Staubli VAL3: XHS3023L1.dtx

public frame fPartReal = {x=0.000, y=0.000, z=0.000, rx=0.000, ry=0.000, rz=0.000, fatherId=world[0]}
public jointRx jtPark = {j1=-10.678, j2=62.119, j3=50.568, j4=-4.773, j5=72.927, j6=-11.595}
public jointRx ptRoutingPath[2001]
  [0] = {j1=-10.678, j2=62.119, j3=50.568, j4=-4.773, j5=72.927, j6=-11.595}
  [1] = {j1=-10.681, j2=62.026, j3=50.659, j4=-4.767, j5=72.852, j6=-11.673}
  [2] = {j1=-10.699, j2=61.483, j3=51.195, j4=-4.725, j5=72.405, j6=-12.130}
  [3] = {j1=-10.720, j2=60.931, j3=51.747, j4=-4.676, j5=71.941, j6=-12.602}
  [4] = {j1=-10.743, j2=60.372, j3=52.310, j4=-4.622, j5=71.468, j6=-13.083}
  [5] = {j1=-10.767, j2=59.811, j3=52.876, j4=-4.565, j5=70.997, j6=-13.564}
  [6] = {j1=-10.793, j2=59.252, j3=53.439, j4=-4.508, j5=70.539, j6=-14.037}
  [7] = {j1=-10.819, j2=58.700, j3=53.990, j4=-4.453, j5=70.102, j6=-14.493}
  [8] = {j1=-10.845, j2=58.158, j3=54.522, j4=-4.401, j5=69.700, j6=-14.925}
  [9] = {j1=-10.866, j2=57.696, j3=54.966, j4=-4.361, j5=69.383, j6=-15.276}
  [10] = {j1=-10.885, j2=57.246, j3=55.388, j4=-4.328, j5=69.100, j6=-15.601}
  [11] = {j1=-10.904, j2=56.809, j3=55.786, j4=-4.299, j5=68.851, j6=-15.902}
  [12] = {j1=-10.922, j2=56.386, j3=56.159, j4=-4.271, j5=68.636, j6=-16.181}
  [13] = {j1=-10.923, j2=56.371, j3=56.172, j4=-4.270, j5=68.629, j6=-16.191}
  [14] = {j1=-10.924, j2=56.416, j3=56.089, j4=-4.262, j5=68.750, j6=-16.121}
  [15] = {j1=-10.923, j2=56.431, j3=56.076, j4=-4.263, j5=68.757, j6=-16.111}
  [16] = {j1=-10.905, j2=56.852, j3=55.709, j4=-4.290, j5=68.965, j6=-15.836}
  [17] = {j1=-10.887, j2=57.285, j3=55.318, j4=-4.319, j5=69.205, j6=-15.540}
  [18] = {j1=-10.868, j2=57.731, j3=54.903, j4=-4.352, j5=69.480, j6=-15.220}
  [19] = {j1=-10.847, j2=58.190, j3=54.465, j4=-4.392, j5=69.790, j6=-14.873}
  [20] = {j1=-10.821, j2=58.729, j3=53.938, j4=-4.443, j5=70.187, j6=-14.445}
  [21] = {j1=-10.795, j2=59.281, j3=53.389, j4=-4.499, j5=70.621, j6=-13.990}
  [22] = {j1=-10.770, j2=59.839, j3=52.827, j4=-4.556, j5=71.079, j6=-13.517}
  [23] = {j1=-10.745, j2=60.400, j3=52.260, j4=-4.612, j5=71.551, j6=-13.035}
  [24] = {j1=-10.722, j2=60.960, j3=51.696, j4=-4.667, j5=72.026, j6=-12.553}
  [25] = {j1=-10.701, j2=61.513, j3=51.143, j4=-4.716, j5=72.492, j6=-12.079}
  [26] = {j1=-10.683, j2=62.055, j3=50.607, j4=-4.758, j5=72.939, j6=-11.621}
  [27] = {j1=-10.681, j2=62.148, j3=50.516, j4=-4.764, j5=73.014, j6=-11.544}
  [28] = {j1=-10.683, j2=62.177, j3=50.465, j4=-4.755, j5=73.100, j6=-11.493}
  [29] = {j1=-10.686, j2=62.084, j3=50.556, j4=-4.748, j5=73.025, j6=-11.570}
  [30] = {j1=-10.704, j2=61.541, j3=51.091, j4=-4.706, j5=72.577, j6=-12.029}
  [31] = {j1=-10.724, j2=60.988, j3=51.645, j4=-4.657, j5=72.110, j6=-12.504}
  [32] = {j1=-10.748, j2=60.428, j3=52.209, j4=-4.603, j5=71.634, j6=-12.987}
  [33] = {j1=-10.772, j2=59.867, j3=52.776, j4=-4.546, j5=71.162, j6=-13.470}
  [34] = {j1=-10.798, j2=59.309, j3=53.338, j4=-4.489, j5=70.704, j6=-13.942}
  [35] = {j1=-10.824, j2=58.759, j3=53.884, j4=-4.434, j5=70.274, j6=-14.396}
  [36] = {j1=-10.849, j2=58.222, j3=54.407, j4=-4.383, j5=69.882, j6=-14.821}
  [37] = {j1=-10.870, j2=57.767, j3=54.839, j4=-4.344, j5=69.580, j6=-15.164}
  [38] = {j1=-10.889, j2=57.325, j3=55.246, j4=-4.311, j5=69.314, j6=-15.478}
  [39] = {j1=-10.907, j2=56.895, j3=55.630, j4=-4.282, j5=69.082, j6=-15.769}
  [40] = {j1=-10.924, j2=56.478, j3=55.991, j4=-4.256, j5=68.881, j6=-16.040}
  [41] = {j1=-10.925, j2=56.463, j3=56.004, j4=-4.255, j5=68.874, j6=-16.050}
  [42] = {j1=-10.926, j2=56.510, j3=55.918, j4=-4.247, j5=68.999, j6=-15.977}
  [43] = {j1=-10.926, j2=56.525, j3=55.906, j4=-4.248, j5=69.006, j6=-15.968}
  [44] = {j1=-10.908, j2=56.939, j3=55.550, j4=-4.274, j5=69.200, j6=-15.701}
  [45] = {j1=-10.891, j2=57.365, j3=55.173, j4=-4.303, j5=69.423, j6=-15.415}
  [46] = {j1=-10.872, j2=57.803, j3=54.773, j4=-4.335, j5=69.680, j6=-15.106}
  [47] = {j1=-10.851, j2=58.255, j3=54.348, j4=-4.374, j5=69.975, j6=-14.768}
  [48] = {j1=-10.826, j2=58.789, j3=53.830, j4=-4.425, j5=70.361, j6=-14.346}
  [49] = {j1=-10.800, j2=59.338, j3=53.286, j4=-4.480, j5=70.788, j6=-13.894}
  [50] = {j1=-10.775, j2=59.896, j3=52.726, j4=-4.537, j5=71.245, j6=-13.422}
  [51] = {j1=-10.750, j2=60.457, j3=52.158, j4=-4.594, j5=71.719, j6=-12.939}
  [52] = {j1=-10.727, j2=61.017, j3=51.593, j4=-4.648, j5=72.196, j6=-12.455}
  [53] = {j1=-10.706, j2=61.571, j3=51.038, j4=-4.697, j5=72.665, j6=-11.979}
  [54] = {j1=-10.688, j2=62.114, j3=50.503, j4=-4.740, j5=73.113, j6=-11.519}
  [55] = {j1=-10.685, j2=62.207, j3=50.412, j4=-4.746, j5=73.189, j6=-11.442}
  [56] = {j1=-10.688, j2=62.236, j3=50.361, j4=-4.737, j5=73.274, j6=-11.391}
  [57] = {j1=-10.690, j2=62.143, j3=50.451, j4=-4.731, j5=73.199, j6=-11.468}
  [58] = {j1=-10.708, j2=61.600, j3=50.987, j4=-4.688, j5=72.750, j6=-11.929}
  [59] = {j1=-10.729, j2=61.046, j3=51.542, j4=-4.639, j5=72.280, j6=-12.406}
  [60] = {j1=-10.752, j2=60.485, j3=52.108, j4=-4.584, j5=71.802, j6=-12.892}
  [61] = {j1=-10.777, j2=59.924, j3=52.675, j4=-4.527, j5=71.329, j6=-13.375}
  [62] = {j1=-10.803, j2=59.367, j3=53.234, j4=-4.471, j5=70.873, j6=-13.847}
  [63] = {j1=-10.828, j2=58.820, j3=53.775, j4=-4.416, j5=70.449, j6=-14.296}
  [64] = {j1=-10.853, j2=58.288, j3=54.287, j4=-4.365, j5=70.069, j6=-14.715}
  [65] = {j1=-10.873, j2=57.840, j3=54.706, j4=-4.327, j5=69.783, j6=-15.048}
  [66] = {j1=-10.892, j2=57.407, j3=55.098, j4=-4.295, j5=69.536, j6=-15.351}
  [67] = {j1=-10.910, j2=56.985, j3=55.467, j4=-4.267, j5=69.322, j6=-15.632}
  [68] = {j1=-10.927, j2=56.575, j3=55.817, j4=-4.241, j5=69.134, j6=-15.895}
  [69] = {j1=-10.927, j2=56.560, j3=55.829, j4=-4.240, j5=69.128, j6=-15.904}
  [70] = {j1=-10.928, j2=56.621, j3=55.718, j4=-4.231, j5=69.288, j6=-15.811}
  [71] = {j1=-10.928, j2=56.636, j3=55.706, j4=-4.232, j5=69.295, j6=-15.802}
  [72] = {j1=-10.911, j2=57.043, j3=55.363, j4=-4.257, j5=69.474, j6=-15.544}
  [73] = {j1=-10.894, j2=57.459, j3=55.003, j4=-4.285, j5=69.677, j6=-15.270}
  [74] = {j1=-10.876, j2=57.887, j3=54.621, j4=-4.317, j5=69.912, j6=-14.974}
  [75] = {j1=-10.856, j2=58.331, j3=54.211, j4=-4.355, j5=70.188, j6=-14.647}
  [76] = {j1=-10.831, j2=58.858, j3=53.705, j4=-4.405, j5=70.560, j6=-14.233}
  [77] = {j1=-10.806, j2=59.403, j3=53.168, j4=-4.459, j5=70.980, j6=-13.786}
  [78] = {j1=-10.780, j2=59.960, j3=52.611, j4=-4.516, j5=71.434, j6=-13.315}
  [79] = {j1=-10.756, j2=60.521, j3=52.043, j4=-4.573, j5=71.908, j6=-12.832}
  [80] = {j1=-10.732, j2=61.082, j3=51.477, j4=-4.627, j5=72.388, j6=-12.345}
  [81] = {j1=-10.711, j2=61.637, j3=50.921, j4=-4.677, j5=72.859, j6=-11.866}
  [82] = {j1=-10.693, j2=62.180, j3=50.385, j4=-4.720, j5=73.309, j6=-11.405}
  [83] = {j1=-10.690, j2=62.273, j3=50.294, j4=-4.726, j5=73.385, j6=-11.327}
  [84] = {j1=-10.678, j2=62.789, j3=49.803, j4=-4.751, j5=73.783, j6=-10.910}
  [85] = {j1=-10.672, j2=63.347, j3=49.311, j4=-4.756, j5=74.142, j6=-10.500}
  [86] = {j1=-10.674, j2=63.830, j3=48.958, j4=-4.737, j5=74.322, j6=-10.212}
  [87] = {j1=-10.676, j2=64.155, j3=48.796, j4=-4.723, j5=74.301, j6=-10.076}
  [88] = {j1=-10.675, j2=64.423, j3=48.741, j4=-4.732, j5=74.135, j6=-10.011}
  [89] = {j1=-10.669, j2=64.639, j3=48.777, j4=-4.763, j5=73.844, j6=-10.010}
  [90] = {j1=-10.658, j2=64.813, j3=48.889, j4=-4.819, j5=73.445, j6=-10.061}
  [91] = {j1=-10.643, j2=64.951, j3=49.062, j4=-4.902, j5=72.957, j6=-10.154}
  [92] = {j1=-10.621, j2=65.058, j3=49.282, j4=-5.014, j5=72.397, j6=-10.276}
  [93] = {j1=-10.593, j2=65.143, j3=49.536, j4=-5.161, j5=71.781, j6=-10.416}
  [94] = {j1=-10.592, j2=65.169, j3=49.489, j4=-5.169, j5=71.871, j6=-10.348}
  [95] = {j1=-10.620, j2=65.085, j3=49.236, j4=-5.021, j5=72.484, j6=-10.211}
  [96] = {j1=-10.642, j2=64.977, j3=49.016, j4=-4.907, j5=73.043, j6=-10.091}
  [97] = {j1=-10.658, j2=64.839, j3=48.843, j4=-4.824, j5=73.530, j6=-10.001}
  [98] = {j1=-10.669, j2=64.666, j3=48.732, j4=-4.766, j5=73.927, j6=-9.952}
  [99] = {j1=-10.675, j2=64.449, j3=48.695, j4=-4.733, j5=74.218, j6=-9.955}
  [100] = {j1=-10.677, j2=64.182, j3=48.749, j4=-4.722, j5=74.384, j6=-10.021}
  [101] = {j1=-10.675, j2=63.857, j3=48.909, j4=-4.734, j5=74.406, j6=-10.160}
  [102] = {j1=-10.673, j2=63.375, j3=49.261, j4=-4.750, j5=74.227, j6=-10.449}
  [103] = {j1=-10.680, j2=62.818, j3=49.751, j4=-4.743, j5=73.869, j6=-10.860}
  [104] = {j1=-10.693, j2=62.303, j3=50.242, j4=-4.718, j5=73.472, j6=-11.278}
  [105] = {j1=-10.695, j2=62.210, j3=50.332, j4=-4.711, j5=73.397, j6=-11.355}
  [106] = {j1=-10.714, j2=61.667, j3=50.868, j4=-4.668, j5=72.946, j6=-11.818}
  [107] = {j1=-10.735, j2=61.112, j3=51.424, j4=-4.618, j5=72.474, j6=-12.297}
  [108] = {j1=-10.758, j2=60.551, j3=51.990, j4=-4.564, j5=71.994, j6=-12.785}
  [109] = {j1=-10.782, j2=59.990, j3=52.557, j4=-4.507, j5=71.521, j6=-13.268}
  [110] = {j1=-10.808, j2=59.434, j3=53.112, j4=-4.451, j5=71.068, j6=-13.738}
  [111] = {j1=-10.833, j2=58.891, j3=53.646, j4=-4.397, j5=70.652, j6=-14.183}
  [112] = {j1=-10.857, j2=58.367, j3=54.146, j4=-4.347, j5=70.288, j6=-14.593}
  [113] = {j1=-10.877, j2=57.927, j3=54.549, j4=-4.310, j5=70.020, j6=-14.915}
  [114] = {j1=-10.895, j2=57.503, j3=54.924, j4=-4.278, j5=69.794, j6=-15.206}
  [115] = {j1=-10.912, j2=57.091, j3=55.276, j4=-4.251, j5=69.600, j6=-15.475}
  [116] = {j1=-10.929, j2=56.687, j3=55.613, j4=-4.226, j5=69.428, j6=-15.729}
  [117] = {j1=-10.929, j2=56.672, j3=55.625, j4=-4.225, j5=69.422, j6=-15.738}
  [118] = {j1=-10.930, j2=56.719, j3=55.540, j4=-4.218, j5=69.545, j6=-15.666}
  [119] = {j1=-10.930, j2=56.734, j3=55.528, j4=-4.219, j5=69.551, j6=-15.657}
  [120] = {j1=-10.913, j2=57.135, j3=55.196, j4=-4.244, j5=69.717, j6=-15.407}
  [121] = {j1=-10.896, j2=57.544, j3=54.850, j4=-4.271, j5=69.904, j6=-15.143}
  [122] = {j1=-10.879, j2=57.964, j3=54.482, j4=-4.302, j5=70.122, j6=-14.856}
  [123] = {j1=-10.859, j2=58.401, j3=54.085, j4=-4.339, j5=70.383, j6=-14.539}
  [124] = {j1=-10.835, j2=58.923, j3=53.589, j4=-4.389, j5=70.742, j6=-14.133}
  [125] = {j1=-10.810, j2=59.465, j3=53.058, j4=-4.442, j5=71.155, j6=-13.690}
  [126] = {j1=-10.785, j2=60.019, j3=52.504, j4=-4.498, j5=71.606, j6=-13.221}
  [127] = {j1=-10.760, j2=60.580, j3=51.938, j4=-4.555, j5=72.079, j6=-12.737}
  [128] = {j1=-10.737, j2=61.141, j3=51.371, j4=-4.609, j5=72.560, j6=-12.250}
  [129] = {j1=-10.716, j2=61.696, j3=50.815, j4=-4.659, j5=73.034, j6=-11.769}
  [130] = {j1=-10.698, j2=62.240, j3=50.279, j4=-4.703, j5=73.485, j6=-11.306}
  [131] = {j1=-10.695, j2=62.333, j3=50.188, j4=-4.709, j5=73.560, j6=-11.228}
  [132] = {j1=-10.682, j2=62.848, j3=49.698, j4=-4.736, j5=73.958, j6=-10.810}
  [133] = {j1=-10.675, j2=63.405, j3=49.209, j4=-4.745, j5=74.315, j6=-10.398}
  [134] = {j1=-10.676, j2=63.886, j3=48.858, j4=-4.731, j5=74.494, j6=-10.107}
  [135] = {j1=-10.677, j2=64.211, j3=48.698, j4=-4.721, j5=74.472, j6=-9.966}
  [136] = {j1=-10.675, j2=64.478, j3=48.644, j4=-4.734, j5=74.307, j6=-9.898}
  [137] = {j1=-10.668, j2=64.695, j3=48.681, j4=-4.769, j5=74.017, j6=-9.893}
  [138] = {j1=-10.657, j2=64.868, j3=48.792, j4=-4.829, j5=73.621, j6=-9.940}
  [139] = {j1=-10.641, j2=65.006, j3=48.965, j4=-4.914, j5=73.136, j6=-10.029}
  [140] = {j1=-10.619, j2=65.114, j3=49.184, j4=-5.029, j5=72.580, j6=-10.147}
  [141] = {j1=-10.590, j2=65.199, j3=49.436, j4=-5.178, j5=71.969, j6=-10.281}
  [142] = {j1=-10.589, j2=65.226, j3=49.390, j4=-5.186, j5=72.057, j6=-10.214}
  [143] = {j1=-10.618, j2=65.140, j3=49.138, j4=-5.036, j5=72.666, j6=-10.082}
  [144] = {j1=-10.640, j2=65.032, j3=48.919, j4=-4.920, j5=73.222, j6=-9.966}
  [145] = {j1=-10.656, j2=64.895, j3=48.746, j4=-4.833, j5=73.706, j6=-9.880}
  [146] = {j1=-10.668, j2=64.721, j3=48.634, j4=-4.772, j5=74.102, j6=-9.835}
  [147] = {j1=-10.675, j2=64.505, j3=48.597, j4=-4.735, j5=74.391, j6=-9.842}
  [148] = {j1=-10.678, j2=64.238, j3=48.650, j4=-4.720, j5=74.556, j6=-9.911}
  [149] = {j1=-10.677, j2=63.914, j3=48.809, j4=-4.727, j5=74.579, j6=-10.054}
  [150] = {j1=-10.677, j2=63.433, j3=49.158, j4=-4.739, j5=74.401, j6=-10.347}
  [151] = {j1=-10.684, j2=62.877, j3=49.646, j4=-4.728, j5=74.044, j6=-10.760}
  [152] = {j1=-10.697, j2=62.362, j3=50.136, j4=-4.701, j5=73.647, j6=-11.179}
  [153] = {j1=-10.700, j2=62.269, j3=50.226, j4=-4.694, j5=73.572, j6=-11.257}
  [154] = {j1=-10.718, j2=61.726, j3=50.761, j4=-4.651, j5=73.121, j6=-11.721}
  [155] = {j1=-10.739, j2=61.171, j3=51.318, j4=-4.601, j5=72.648, j6=-12.202}
  [156] = {j1=-10.762, j2=60.611, j3=51.883, j4=-4.546, j5=72.168, j6=-12.690}
  [157] = {j1=-10.787, j2=60.050, j3=52.448, j4=-4.490, j5=71.696, j6=-13.173}
  [158] = {j1=-10.812, j2=59.497, j3=53.000, j4=-4.434, j5=71.247, j6=-13.641}
  [159] = {j1=-10.837, j2=58.957, j3=53.527, j4=-4.381, j5=70.838, j6=-14.082}
  [160] = {j1=-10.861, j2=58.438, j3=54.018, j4=-4.332, j5=70.485, j6=-14.484}
  [161] = {j1=-10.880, j2=58.005, j3=54.409, j4=-4.295, j5=70.232, j6=-14.797}
  [162] = {j1=-10.897, j2=57.588, j3=54.770, j4=-4.264, j5=70.022, j6=-15.079}
  [163] = {j1=-10.914, j2=57.183, j3=55.110, j4=-4.237, j5=69.842, j6=-15.340}
  [164] = {j1=-10.930, j2=56.784, j3=55.437, j4=-4.213, j5=69.681, j6=-15.587}
  [165] = {j1=-10.931, j2=56.770, j3=55.449, j4=-4.212, j5=69.676, j6=-15.596}
  [166] = {j1=-10.932, j2=56.814, j3=55.368, j4=-4.205, j5=69.793, j6=-15.527}
  [167] = {j1=-10.931, j2=56.829, j3=55.356, j4=-4.206, j5=69.799, j6=-15.518}
  [168] = {j1=-10.915, j2=57.225, j3=55.032, j4=-4.231, j5=69.956, j6=-15.273}
  [169] = {j1=-10.899, j2=57.628, j3=54.698, j4=-4.258, j5=70.130, j6=-15.017}
  [170] = {j1=-10.881, j2=58.042, j3=54.342, j4=-4.288, j5=70.334, j6=-14.739}
  [171] = {j1=-10.862, j2=58.473, j3=53.955, j4=-4.325, j5=70.582, j6=-14.429}
  [172] = {j1=-10.839, j2=58.990, j3=53.469, j4=-4.373, j5=70.930, j6=-14.030}
  [173] = {j1=-10.814, j2=59.528, j3=52.944, j4=-4.426, j5=71.336, j6=-13.592}
  [174] = {j1=-10.789, j2=60.081, j3=52.394, j4=-4.481, j5=71.783, j6=-13.125}
  [175] = {j1=-10.765, j2=60.641, j3=51.830, j4=-4.537, j5=72.255, j6=-12.642}
  [176] = {j1=-10.741, j2=61.201, j3=51.264, j4=-4.592, j5=72.735, j6=-12.154}
  [177] = {j1=-10.720, j2=61.756, j3=50.708, j4=-4.642, j5=73.209, j6=-11.672}
  [178] = {j1=-10.702, j2=62.299, j3=50.173, j4=-4.686, j5=73.660, j6=-11.208}
  [179] = {j1=-10.699, j2=62.392, j3=50.082, j4=-4.693, j5=73.736, j6=-11.130}
  [180] = {j1=-10.686, j2=62.907, j3=49.593, j4=-4.721, j5=74.133, j6=-10.710}
  [181] = {j1=-10.678, j2=63.464, j3=49.105, j4=-4.733, j5=74.490, j6=-10.296}
  [182] = {j1=-10.678, j2=63.944, j3=48.756, j4=-4.725, j5=74.668, j6=-10.000}
  [183] = {j1=-10.678, j2=64.268, j3=48.597, j4=-4.720, j5=74.646, j6=-9.856}
  [184] = {j1=-10.675, j2=64.535, j3=48.545, j4=-4.737, j5=74.482, j6=-9.785}
  [185] = {j1=-10.667, j2=64.751, j3=48.582, j4=-4.776, j5=74.193, j6=-9.776}
  [186] = {j1=-10.655, j2=64.924, j3=48.694, j4=-4.838, j5=73.799, j6=-9.819}
  [187] = {j1=-10.639, j2=65.062, j3=48.867, j4=-4.927, j5=73.316, j6=-9.904}
  [188] = {j1=-10.616, j2=65.170, j3=49.085, j4=-5.044, j5=72.763, j6=-10.018}
  [189] = {j1=-10.587, j2=65.256, j3=49.337, j4=-5.196, j5=72.156, j6=-10.148}
  [190] = {j1=-10.586, j2=65.282, j3=49.292, j4=-5.204, j5=72.243, j6=-10.082}
  [191] = {j1=-10.615, j2=65.196, j3=49.040, j4=-5.051, j5=72.849, j6=-9.954}
  [192] = {j1=-10.638, j2=65.088, j3=48.821, j4=-4.932, j5=73.402, j6=-9.842}
  [193] = {j1=-10.655, j2=64.951, j3=48.648, j4=-4.843, j5=73.884, j6=-9.759}
  [194] = {j1=-10.667, j2=64.778, j3=48.535, j4=-4.779, j5=74.278, j6=-9.717}
  [195] = {j1=-10.675, j2=64.562, j3=48.497, j4=-4.738, j5=74.567, j6=-9.728}
  [196] = {j1=-10.679, j2=64.296, j3=48.549, j4=-4.719, j5=74.731, j6=-9.801}
  [197] = {j1=-10.679, j2=63.972, j3=48.706, j4=-4.721, j5=74.753, j6=-9.947}
  [198] = {j1=-10.680, j2=63.492, j3=49.054, j4=-4.728, j5=74.576, j6=-10.245}
  [199] = {j1=-10.688, j2=62.936, j3=49.541, j4=-4.714, j5=74.219, j6=-10.661}
  [200] = {j1=-10.701, j2=62.422, j3=50.030, j4=-4.685, j5=73.823, j6=-11.081}
  [201] = {j1=-10.704, j2=62.329, j3=50.120, j4=-4.678, j5=73.748, j6=-11.160}
  [202] = {j1=-10.723, j2=61.787, j3=50.654, j4=-4.634, j5=73.297, j6=-11.624}
  [203] = {j1=-10.744, j2=61.232, j3=51.210, j4=-4.583, j5=72.824, j6=-12.106}
  [204] = {j1=-10.767, j2=60.672, j3=51.774, j4=-4.529, j5=72.344, j6=-12.594}
  [205] = {j1=-10.791, j2=60.113, j3=52.336, j4=-4.473, j5=71.874, j6=-13.076}
  [206] = {j1=-10.816, j2=59.562, j3=52.884, j4=-4.418, j5=71.430, j6=-13.542}
  [207] = {j1=-10.840, j2=59.025, j3=53.405, j4=-4.366, j5=71.028, j6=-13.978}
  [208] = {j1=-10.864, j2=58.511, j3=53.886, j4=-4.318, j5=70.686, j6=-14.374}
  [209] = {j1=-10.883, j2=58.083, j3=54.268, j4=-4.282, j5=70.444, j6=-14.680}
  [210] = {j1=-10.900, j2=57.672, j3=54.618, j4=-4.252, j5=70.247, j6=-14.955}
  [211] = {j1=-10.916, j2=57.272, j3=54.948, j4=-4.225, j5=70.079, j6=-15.208}
  [212] = {j1=-10.932, j2=56.878, j3=55.267, j4=-4.201, j5=69.926, j6=-15.451}
  [213] = {j1=-10.932, j2=56.864, j3=55.279, j4=-4.200, j5=69.921, j6=-15.460}
  [214] = {j1=-10.933, j2=56.906, j3=55.202, j4=-4.193, j5=70.034, j6=-15.393}
  [215] = {j1=-10.933, j2=56.921, j3=55.190, j4=-4.194, j5=70.039, j6=-15.385}
  [216] = {j1=-10.917, j2=57.314, j3=54.873, j4=-4.218, j5=70.189, j6=-15.144}
  [217] = {j1=-10.901, j2=57.711, j3=54.547, j4=-4.245, j5=70.353, j6=-14.893}
  [218] = {j1=-10.884, j2=58.120, j3=54.200, j4=-4.275, j5=70.546, j6=-14.621}
  [219] = {j1=-10.865, j2=58.546, j3=53.823, j4=-4.310, j5=70.784, j6=-14.318}
  [220] = {j1=-10.842, j2=59.059, j3=53.345, j4=-4.358, j5=71.122, j6=-13.925}
  [221] = {j1=-10.818, j2=59.594, j3=52.827, j4=-4.409, j5=71.521, j6=-13.491}
  [222] = {j1=-10.793, j2=60.144, j3=52.281, j4=-4.464, j5=71.963, j6=-13.027}
  [223] = {j1=-10.769, j2=60.702, j3=51.720, j4=-4.520, j5=72.432, j6=-12.546}
  [224] = {j1=-10.746, j2=61.262, j3=51.156, j4=-4.575, j5=72.911, j6=-12.058}
  [225] = {j1=-10.725, j2=61.816, j3=50.601, j4=-4.625, j5=73.384, j6=-11.576}
  [226] = {j1=-10.706, j2=62.359, j3=50.066, j4=-4.670, j5=73.836, j6=-11.111}
  [227] = {j1=-10.703, j2=62.452, j3=49.976, j4=-4.677, j5=73.911, j6=-11.033}
  [228] = {j1=-10.690, j2=62.966, j3=49.488, j4=-4.707, j5=74.308, j6=-10.611}
  [229] = {j1=-10.681, j2=63.523, j3=49.001, j4=-4.722, j5=74.666, j6=-10.194}
  [230] = {j1=-10.679, j2=64.003, j3=48.653, j4=-4.719, j5=74.844, j6=-9.894}
  [231] = {j1=-10.679, j2=64.326, j3=48.495, j4=-4.719, j5=74.823, j6=-9.746}
  [232] = {j1=-10.675, j2=64.592, j3=48.444, j4=-4.740, j5=74.659, j6=-9.671}
  [233] = {j1=-10.666, j2=64.808, j3=48.482, j4=-4.782, j5=74.371, j6=-9.658}
  [234] = {j1=-10.654, j2=64.981, j3=48.595, j4=-4.848, j5=73.978, j6=-9.698}
  [235] = {j1=-10.637, j2=65.118, j3=48.768, j4=-4.939, j5=73.497, j6=-9.779}
  [236] = {j1=-10.614, j2=65.227, j3=48.987, j4=-5.059, j5=72.946, j6=-9.890}
  [237] = {j1=-10.584, j2=65.312, j3=49.239, j4=-5.213, j5=72.342, j6=-10.017}
  [238] = {j1=-10.583, j2=65.337, j3=49.194, j4=-5.221, j5=72.428, j6=-9.951}
  [239] = {j1=-10.612, j2=65.252, j3=48.942, j4=-5.066, j5=73.031, j6=-9.826}
  [240] = {j1=-10.636, j2=65.144, j3=48.722, j4=-4.945, j5=73.582, j6=-9.717}
  [241] = {j1=-10.653, j2=65.008, j3=48.548, j4=-4.852, j5=74.063, j6=-9.638}
  [242] = {j1=-10.666, j2=64.835, j3=48.435, j4=-4.785, j5=74.456, j6=-9.600}
  [243] = {j1=-10.675, j2=64.620, j3=48.395, j4=-4.741, j5=74.744, j6=-9.614}
  [244] = {j1=-10.679, j2=64.354, j3=48.446, j4=-4.718, j5=74.908, j6=-9.691}
  [245] = {j1=-10.680, j2=64.031, j3=48.603, j4=-4.716, j5=74.930, j6=-9.840}
  [246] = {j1=-10.683, j2=63.551, j3=48.950, j4=-4.717, j5=74.751, j6=-10.143}
  [247] = {j1=-10.692, j2=62.995, j3=49.436, j4=-4.699, j5=74.394, j6=-10.562}
  [248] = {j1=-10.706, j2=62.481, j3=49.924, j4=-4.669, j5=73.998, j6=-10.984}
  [249] = {j1=-10.708, j2=62.389, j3=50.014, j4=-4.662, j5=73.923, j6=-11.063}
  [250] = {j1=-10.727, j2=61.847, j3=50.547, j4=-4.617, j5=73.472, j6=-11.528}
  [251] = {j1=-10.748, j2=61.293, j3=51.101, j4=-4.566, j5=73.000, j6=-12.010}
  [252] = {j1=-10.771, j2=60.734, j3=51.663, j4=-4.512, j5=72.523, j6=-12.497}
  [253] = {j1=-10.795, j2=60.177, j3=52.221, j4=-4.456, j5=72.057, j6=-12.977}
  [254] = {j1=-10.820, j2=59.628, j3=52.764, j4=-4.402, j5=71.618, j6=-13.440}
  [255] = {j1=-10.844, j2=59.095, j3=53.279, j4=-4.350, j5=71.223, j6=-13.872}
  [256] = {j1=-10.867, j2=58.585, j3=53.753, j4=-4.304, j5=70.889, j6=-14.262}
  [257] = {j1=-10.885, j2=58.161, j3=54.126, j4=-4.269, j5=70.656, j6=-14.563}
  [258] = {j1=-10.902, j2=57.755, j3=54.469, j4=-4.239, j5=70.468, j6=-14.832}
  [259] = {j1=-10.918, j2=57.359, j3=54.791, j4=-4.213, j5=70.309, j6=-15.080}
  [260] = {j1=-10.933, j2=56.968, j3=55.105, j4=-4.189, j5=70.162, j6=-15.320}
  [261] = {j1=-10.934, j2=56.954, j3=55.116, j4=-4.188, j5=70.157, j6=-15.329}
  [262] = {j1=-10.935, j2=56.995, j3=55.043, j4=-4.181, j5=70.265, j6=-15.265}
  [263] = {j1=-10.934, j2=57.009, j3=55.031, j4=-4.182, j5=70.270, j6=-15.257}
  [264] = {j1=-10.919, j2=57.399, j3=54.719, j4=-4.207, j5=70.416, j6=-15.018}
  [265] = {j1=-10.903, j2=57.794, j3=54.399, j4=-4.233, j5=70.573, j6=-14.771}
  [266] = {j1=-10.886, j2=58.199, j3=54.059, j4=-4.262, j5=70.758, j6=-14.504}
  [267] = {j1=-10.868, j2=58.621, j3=53.689, j4=-4.297, j5=70.988, j6=-14.206}
  [268] = {j1=-10.846, j2=59.130, j3=53.218, j4=-4.343, j5=71.318, j6=-13.818}
  [269] = {j1=-10.822, j2=59.661, j3=52.705, j4=-4.394, j5=71.711, j6=-13.388}
  [270] = {j1=-10.797, j2=60.209, j3=52.164, j4=-4.448, j5=72.148, j6=-12.927}
  [271] = {j1=-10.773, j2=60.765, j3=51.607, j4=-4.503, j5=72.612, j6=-12.448}
  [272] = {j1=-10.750, j2=61.323, j3=51.047, j4=-4.558, j5=73.088, j6=-11.962}
  [273] = {j1=-10.729, j2=61.877, j3=50.494, j4=-4.609, j5=73.559, j6=-11.480}
  [274] = {j1=-10.711, j2=62.419, j3=49.961, j4=-4.654, j5=74.010, j6=-11.015}
  [275] = {j1=-10.708, j2=62.512, j3=49.870, j4=-4.661, j5=74.086, j6=-10.936}
  [276] = {j1=-10.694, j2=63.026, j3=49.383, j4=-4.692, j5=74.483, j6=-10.513}
  [277] = {j1=-10.684, j2=63.582, j3=48.896, j4=-4.711, j5=74.841, j6=-10.092}
  [278] = {j1=-10.681, j2=64.062, j3=48.549, j4=-4.713, j5=75.021, j6=-9.787}
  [279] = {j1=-10.680, j2=64.385, j3=48.392, j4=-4.718, j5=75.000, j6=-9.635}
  [280] = {j1=-10.675, j2=64.651, j3=48.341, j4=-4.743, j5=74.837, j6=-9.556}
  [281] = {j1=-10.666, j2=64.866, j3=48.381, j4=-4.789, j5=74.550, j6=-9.541}
  [282] = {j1=-10.652, j2=65.038, j3=48.495, j4=-4.858, j5=74.158, j6=-9.577}
  [283] = {j1=-10.634, j2=65.175, j3=48.669, j4=-4.952, j5=73.678, j6=-9.656}
  [284] = {j1=-10.611, j2=65.283, j3=48.889, j4=-5.074, j5=73.128, j6=-9.763}
  [285] = {j1=-10.581, j2=65.368, j3=49.141, j4=-5.230, j5=72.526, j6=-9.886}
  [286] = {j1=-10.580, j2=65.393, j3=49.098, j4=-5.238, j5=72.611, j6=-9.822}
  [287] = {j1=-10.610, j2=65.308, j3=48.844, j4=-5.081, j5=73.213, j6=-9.700}
  [288] = {j1=-10.634, j2=65.201, j3=48.623, j4=-4.957, j5=73.763, j6=-9.594}
  [289] = {j1=-10.652, j2=65.065, j3=48.448, j4=-4.862, j5=74.243, j6=-9.517}
  [290] = {j1=-10.665, j2=64.893, j3=48.333, j4=-4.792, j5=74.636, j6=-9.481}
  [291] = {j1=-10.675, j2=64.678, j3=48.292, j4=-4.744, j5=74.923, j6=-9.499}
  [292] = {j1=-10.680, j2=64.414, j3=48.342, j4=-4.717, j5=75.087, j6=-9.579}
  [293] = {j1=-10.682, j2=64.090, j3=48.498, j4=-4.710, j5=75.107, j6=-9.733}
  [294] = {j1=-10.686, j2=63.610, j3=48.845, j4=-4.706, j5=74.927, j6=-10.041}
  [295] = {j1=-10.696, j2=63.055, j3=49.331, j4=-4.685, j5=74.569, j6=-10.464}
  [296] = {j1=-10.710, j2=62.541, j3=49.818, j4=-4.653, j5=74.172, j6=-10.888}
  [297] = {j1=-10.713, j2=62.448, j3=49.908, j4=-4.646, j5=74.097, j6=-10.967}
  [298] = {j1=-10.731, j2=61.907, j3=50.440, j4=-4.600, j5=73.647, j6=-11.432}
  [299] = {j1=-10.752, j2=61.355, j3=50.991, j4=-4.549, j5=73.178, j6=-11.914}
  [300] = {j1=-10.775, j2=60.798, j3=51.549, j4=-4.495, j5=72.705, j6=-12.399}
  [301] = {j1=-10.799, j2=60.243, j3=52.104, j4=-4.440, j5=72.243, j6=-12.877}
  [302] = {j1=-10.823, j2=59.697, j3=52.642, j4=-4.386, j5=71.810, j6=-13.336}
  [303] = {j1=-10.847, j2=59.167, j3=53.151, j4=-4.336, j5=71.421, j6=-13.764}
  [304] = {j1=-10.869, j2=58.660, j3=53.618, j4=-4.290, j5=71.095, j6=-14.149}
  [305] = {j1=-10.887, j2=58.240, j3=53.985, j4=-4.256, j5=70.868, j6=-14.446}
  [306] = {j1=-10.904, j2=57.837, j3=54.321, j4=-4.227, j5=70.687, j6=-14.711}
  [307] = {j1=-10.920, j2=57.444, j3=54.639, j4=-4.201, j5=70.532, j6=-14.956}
  [308] = {j1=-10.935, j2=57.054, j3=54.949, j4=-4.177, j5=70.389, j6=-15.194}
  [309] = {j1=-10.936, j2=57.040, j3=54.960, j4=-4.176, j5=70.384, j6=-15.203}
  [310] = {j1=-10.937, j2=57.079, j3=54.891, j4=-4.170, j5=70.487, j6=-15.143}
  [311] = {j1=-10.936, j2=57.093, j3=54.879, j4=-4.171, j5=70.492, j6=-15.134}
  [312] = {j1=-10.921, j2=57.482, j3=54.569, j4=-4.195, j5=70.636, j6=-14.896}
  [313] = {j1=-10.905, j2=57.875, j3=54.253, j4=-4.221, j5=70.789, j6=-14.651}
  [314] = {j1=-10.889, j2=58.277, j3=53.918, j4=-4.250, j5=70.970, j6=-14.387}
  [315] = {j1=-10.871, j2=58.697, j3=53.553, j4=-4.283, j5=71.194, j6=-14.093}
  [316] = {j1=-10.849, j2=59.202, j3=53.088, j4=-4.328, j5=71.518, j6=-13.709}
  [317] = {j1=-10.825, j2=59.731, j3=52.581, j4=-4.378, j5=71.904, j6=-13.283}
  [318] = {j1=-10.801, j2=60.275, j3=52.045, j4=-4.432, j5=72.335, j6=-12.826}
  [319] = {j1=-10.777, j2=60.829, j3=51.493, j4=-4.487, j5=72.794, j6=-12.349}
  [320] = {j1=-10.755, j2=61.385, j3=50.937, j4=-4.541, j5=73.266, j6=-11.865}
  [321] = {j1=-10.733, j2=61.937, j3=50.387, j4=-4.592, j5=73.734, j6=-11.385}
  [322] = {j1=-10.715, j2=62.478, j3=49.856, j4=-4.637, j5=74.184, j6=-10.919}
  [323] = {j1=-10.712, j2=62.571, j3=49.765, j4=-4.645, j5=74.259, j6=-10.841}
  [324] = {j1=-10.698, j2=63.085, j3=49.278, j4=-4.677, j5=74.657, j6=-10.415}
  [325] = {j1=-10.687, j2=63.641, j3=48.791, j4=-4.700, j5=75.017, j6=-9.990}
  [326] = {j1=-10.683, j2=64.121, j3=48.444, j4=-4.707, j5=75.199, j6=-9.680}
  [327] = {j1=-10.680, j2=64.445, j3=48.287, j4=-4.716, j5=75.179, j6=-9.524}
  [328] = {j1=-10.674, j2=64.710, j3=48.238, j4=-4.746, j5=75.017, j6=-9.441}
  [329] = {j1=-10.665, j2=64.924, j3=48.279, j4=-4.795, j5=74.730, j6=-9.422}
  [330] = {j1=-10.651, j2=65.095, j3=48.395, j4=-4.867, j5=74.338, j6=-9.456}
  [331] = {j1=-10.632, j2=65.231, j3=48.570, j4=-4.964, j5=73.858, j6=-9.532}
  [332] = {j1=-10.608, j2=65.338, j3=48.791, j4=-5.089, j5=73.310, j6=-9.637}
  [333] = {j1=-10.578, j2=65.423, j3=49.045, j4=-5.247, j5=72.709, j6=-9.758}
  [334] = {j1=-10.577, j2=65.447, j3=49.002, j4=-5.255, j5=72.793, j6=-9.694}
  [335] = {j1=-10.607, j2=65.363, j3=48.747, j4=-5.096, j5=73.394, j6=-9.574}
  [336] = {j1=-10.631, j2=65.257, j3=48.525, j4=-4.970, j5=73.943, j6=-9.470}
  [337] = {j1=-10.650, j2=65.122, j3=48.348, j4=-4.872, j5=74.423, j6=-9.396}
  [338] = {j1=-10.664, j2=64.951, j3=48.231, j4=-4.798, j5=74.816, j6=-9.363}
  [339] = {j1=-10.674, j2=64.738, j3=48.189, j4=-4.747, j5=75.103, j6=-9.383}
  [340] = {j1=-10.681, j2=64.473, j3=48.237, j4=-4.715, j5=75.266, j6=-9.468}
  [341] = {j1=-10.684, j2=64.150, j3=48.393, j4=-4.704, j5=75.285, j6=-9.626}
  [342] = {j1=-10.689, j2=63.670, j3=48.741, j4=-4.695, j5=75.103, j6=-9.939}
  [343] = {j1=-10.700, j2=63.113, j3=49.227, j4=-4.670, j5=74.742, j6=-10.367}
  [344] = {j1=-10.714, j2=62.600, j3=49.714, j4=-4.637, j5=74.345, j6=-10.793}
  [345] = {j1=-10.717, j2=62.507, j3=49.803, j4=-4.629, j5=74.270, j6=-10.872}
  [346] = {j1=-10.736, j2=61.967, j3=50.333, j4=-4.584, j5=73.822, j6=-11.337}
  [347] = {j1=-10.757, j2=61.416, j3=50.881, j4=-4.533, j5=73.356, j6=-11.817}
  [348] = {j1=-10.779, j2=60.862, j3=51.435, j4=-4.478, j5=72.888, j6=-12.299}
  [349] = {j1=-10.803, j2=60.310, j3=51.983, j4=-4.424, j5=72.432, j6=-12.774}
  [350] = {j1=-10.827, j2=59.767, j3=52.516, j4=-4.371, j5=72.005, j6=-13.229}
  [351] = {j1=-10.850, j2=59.240, j3=53.019, j4=-4.321, j5=71.623, j6=-13.653}
  [352] = {j1=-10.872, j2=58.737, j3=53.481, j4=-4.277, j5=71.302, j6=-14.035}
  [353] = {j1=-10.890, j2=58.318, j3=53.844, j4=-4.244, j5=71.080, j6=-14.329}
  [354] = {j1=-10.906, j2=57.917, j3=54.177, j4=-4.216, j5=70.901, j6=-14.592}
  [355] = {j1=-10.922, j2=57.525, j3=54.492, j4=-4.190, j5=70.749, j6=-14.837}
  [356] = {j1=-10.937, j2=57.137, j3=54.801, j4=-4.166, j5=70.606, j6=-15.075}
  [357] = {j1=-10.937, j2=57.122, j3=54.812, j4=-4.165, j5=70.601, j6=-15.083}
  [358] = {j1=-10.939, j2=57.159, j3=54.747, j4=-4.159, j5=70.699, j6=-15.026}
  [359] = {j1=-10.938, j2=57.173, j3=54.735, j4=-4.160, j5=70.704, j6=-15.017}
  [360] = {j1=-10.923, j2=57.562, j3=54.425, j4=-4.184, j5=70.848, j6=-14.779}
  [361] = {j1=-10.907, j2=57.954, j3=54.110, j4=-4.209, j5=71.001, j6=-14.534}
  [362] = {j1=-10.891, j2=58.355, j3=53.777, j4=-4.237, j5=71.180, j6=-14.271}
  [363] = {j1=-10.874, j2=58.773, j3=53.415, j4=-4.270, j5=71.402, j6=-13.978}
  [364] = {j1=-10.852, j2=59.276, j3=52.955, j4=-4.314, j5=71.721, j6=-13.597}
  [365] = {j1=-10.829, j2=59.802, j3=52.454, j4=-4.363, j5=72.101, j6=-13.175}
  [366] = {j1=-10.805, j2=60.343, j3=51.924, j4=-4.416, j5=72.525, j6=-12.722}
  [367] = {j1=-10.781, j2=60.894, j3=51.378, j4=-4.470, j5=72.978, j6=-12.249}
  [368] = {j1=-10.759, j2=61.447, j3=50.826, j4=-4.524, j5=73.444, j6=-11.768}
  [369] = {j1=-10.738, j2=61.997, j3=50.280, j4=-4.576, j5=73.909, j6=-11.289}
  [370] = {j1=-10.719, j2=62.537, j3=49.751, j4=-4.621, j5=74.356, j6=-10.824}
  [371] = {j1=-10.716, j2=62.629, j3=49.661, j4=-4.629, j5=74.431, j6=-10.745}
  [372] = {j1=-10.702, j2=63.143, j3=49.174, j4=-4.663, j5=74.830, j6=-10.318}
  [373] = {j1=-10.690, j2=63.700, j3=48.687, j4=-4.689, j5=75.193, j6=-9.888}
  [374] = {j1=-10.685, j2=64.181, j3=48.338, j4=-4.701, j5=75.377, j6=-9.572}
  [375] = {j1=-10.681, j2=64.504, j3=48.182, j4=-4.715, j5=75.359, j6=-9.412}
  [376] = {j1=-10.674, j2=64.769, j3=48.134, j4=-4.748, j5=75.197, j6=-9.326}
  [377] = {j1=-10.664, j2=64.982, j3=48.176, j4=-4.802, j5=74.910, j6=-9.304}
  [378] = {j1=-10.649, j2=65.153, j3=48.294, j4=-4.877, j5=74.518, j6=-9.335}
  [379] = {j1=-10.630, j2=65.287, j3=48.472, j4=-4.977, j5=74.039, j6=-9.409}
  [380] = {j1=-10.606, j2=65.393, j3=48.695, j4=-5.104, j5=73.490, j6=-9.512}
  [381] = {j1=-10.575, j2=65.477, j3=48.950, j4=-5.264, j5=72.889, j6=-9.631}
  [382] = {j1=-10.574, j2=65.501, j3=48.908, j4=-5.272, j5=72.972, j6=-9.568}
  [383] = {j1=-10.605, j2=65.418, j3=48.651, j4=-5.111, j5=73.573, j6=-9.449}
  [384] = {j1=-10.629, j2=65.313, j3=48.426, j4=-4.982, j5=74.123, j6=-9.347}
  [385] = {j1=-10.649, j2=65.180, j3=48.247, j4=-4.882, j5=74.603, j6=-9.275}
  [386] = {j1=-10.663, j2=65.010, j3=48.128, j4=-4.805, j5=74.997, j6=-9.244}
  [387] = {j1=-10.674, j2=64.797, j3=48.084, j4=-4.750, j5=75.284, j6=-9.268}
  [388] = {j1=-10.682, j2=64.533, j3=48.132, j4=-4.714, j5=75.446, j6=-9.355}
  [389] = {j1=-10.686, j2=64.210, j3=48.287, j4=-4.698, j5=75.464, j6=-9.518}
  [390] = {j1=-10.692, j2=63.729, j3=48.636, j4=-4.683, j5=75.279, j6=-9.837}
  [391] = {j1=-10.704, j2=63.172, j3=49.124, j4=-4.656, j5=74.915, j6=-10.270}
  [392] = {j1=-10.718, j2=62.658, j3=49.610, j4=-4.621, j5=74.516, j6=-10.698}
  [393] = {j1=-10.721, j2=62.566, j3=49.699, j4=-4.613, j5=74.442, j6=-10.777}
  [394] = {j1=-10.740, j2=62.027, j3=50.227, j4=-4.567, j5=73.996, j6=-11.242}
  [395] = {j1=-10.761, j2=61.479, j3=50.770, j4=-4.516, j5=73.535, j6=-11.719}
  [396] = {j1=-10.783, j2=60.927, j3=51.318, j4=-4.462, j5=73.073, j6=-12.199}
  [397] = {j1=-10.807, j2=60.379, j3=51.861, j4=-4.408, j5=72.624, j6=-12.669}
  [398] = {j1=-10.830, j2=59.839, j3=52.387, j4=-4.356, j5=72.204, j6=-13.120}
  [399] = {j1=-10.853, j2=59.315, j3=52.885, j4=-4.307, j5=71.827, j6=-13.541}
  [400] = {j1=-10.875, j2=58.814, j3=53.342, j4=-4.264, j5=71.510, j6=-13.920}
  [401] = {j1=-10.892, j2=58.396, j3=53.704, j4=-4.232, j5=71.290, j6=-14.212}
  [402] = {j1=-10.908, j2=57.995, j3=54.036, j4=-4.204, j5=71.111, j6=-14.476}
  [403] = {j1=-10.923, j2=57.604, j3=54.351, j4=-4.179, j5=70.957, j6=-14.721}
  [404] = {j1=-10.939, j2=57.215, j3=54.661, j4=-4.155, j5=70.813, j6=-14.961}
  [405] = {j1=-10.939, j2=57.200, j3=54.672, j4=-4.154, j5=70.808, j6=-14.969}
  [406] = {j1=-10.941, j2=57.235, j3=54.610, j4=-4.148, j5=70.901, j6=-14.915}
  [407] = {j1=-10.940, j2=57.249, j3=54.598, j4=-4.149, j5=70.906, j6=-14.906}
  [408] = {j1=-10.925, j2=57.639, j3=54.287, j4=-4.173, j5=71.053, j6=-14.665}
  [409] = {j1=-10.909, j2=58.032, j3=53.971, j4=-4.198, j5=71.209, j6=-14.418}
  [410] = {j1=-10.893, j2=58.433, j3=53.637, j4=-4.225, j5=71.390, j6=-14.155}
  [411] = {j1=-10.876, j2=58.851, j3=53.276, j4=-4.257, j5=71.611, j6=-13.862}
  [412] = {j1=-10.855, j2=59.352, j3=52.819, j4=-4.300, j5=71.927, j6=-13.484}
  [413] = {j1=-10.832, j2=59.875, j3=52.323, j4=-4.348, j5=72.302, j6=-13.065}
  [414] = {j1=-10.809, j2=60.413, j3=51.800, j4=-4.400, j5=72.719, j6=-12.616}
  [415] = {j1=-10.785, j2=60.960, j3=51.260, j4=-4.454, j5=73.164, j6=-12.148}
  [416] = {j1=-10.763, j2=61.510, j3=50.715, j4=-4.508, j5=73.624, j6=-11.670}
  [417] = {j1=-10.742, j2=62.057, j3=50.174, j4=-4.559, j5=74.083, j6=-11.194}
  [418] = {j1=-10.723, j2=62.595, j3=49.647, j4=-4.605, j5=74.528, j6=-10.729}
  [419] = {j1=-10.720, j2=62.688, j3=49.558, j4=-4.613, j5=74.603, j6=-10.651}
  [420] = {j1=-10.706, j2=63.202, j3=49.071, j4=-4.649, j5=75.003, j6=-10.221}
  [421] = {j1=-10.693, j2=63.760, j3=48.582, j4=-4.678, j5=75.368, j6=-9.786}
  [422] = {j1=-10.687, j2=64.241, j3=48.232, j4=-4.695, j5=75.556, j6=-9.464}
  [423] = {j1=-10.682, j2=64.565, j3=48.076, j4=-4.714, j5=75.539, j6=-9.299}
  [424] = {j1=-10.674, j2=64.829, j3=48.029, j4=-4.751, j5=75.378, j6=-9.210}
  [425] = {j1=-10.663, j2=65.041, j3=48.073, j4=-4.808, j5=75.091, j6=-9.185}
  [426] = {j1=-10.648, j2=65.210, j3=48.193, j4=-4.887, j5=74.698, j6=-9.214}
  [427] = {j1=-10.628, j2=65.344, j3=48.374, j4=-4.989, j5=74.218, j6=-9.286}
  [428] = {j1=-10.603, j2=65.448, j3=48.599, j4=-5.119, j5=73.668, j6=-9.387}
  [429] = {j1=-10.572, j2=65.530, j3=48.857, j4=-5.281, j5=73.067, j6=-9.505}
  [430] = {j1=-10.571, j2=65.554, j3=48.816, j4=-5.289, j5=73.149, j6=-9.443}
  [431] = {j1=-10.602, j2=65.473, j3=48.556, j4=-5.126, j5=73.751, j6=-9.325}
  [432] = {j1=-10.627, j2=65.369, j3=48.329, j4=-4.995, j5=74.302, j6=-9.225}
  [433] = {j1=-10.647, j2=65.237, j3=48.147, j4=-4.891, j5=74.784, j6=-9.154}
  [434] = {j1=-10.662, j2=65.069, j3=48.025, j4=-4.811, j5=75.178, j6=-9.126}
  [435] = {j1=-10.674, j2=64.857, j3=47.979, j4=-4.752, j5=75.465, j6=-9.151}
  [436] = {j1=-10.682, j2=64.594, j3=48.026, j4=-4.713, j5=75.627, j6=-9.243}
  [437] = {j1=-10.688, j2=64.270, j3=48.181, j4=-4.692, j5=75.643, j6=-9.410}
  [438] = {j1=-10.695, j2=63.788, j3=48.531, j4=-4.672, j5=75.454, j6=-9.735}
  [439] = {j1=-10.708, j2=63.230, j3=49.020, j4=-4.641, j5=75.087, j6=-10.173}
  [440] = {j1=-10.722, j2=62.717, j3=49.507, j4=-4.605, j5=74.687, j6=-10.603}
  [441] = {j1=-10.725, j2=62.624, j3=49.596, j4=-4.597, j5=74.613, j6=-10.682}
  [442] = {j1=-10.744, j2=62.087, j3=50.120, j4=-4.551, j5=74.170, j6=-11.146}
  [443] = {j1=-10.765, j2=61.542, j3=50.658, j4=-4.500, j5=73.715, j6=-11.621}
  [444] = {j1=-10.787, j2=60.994, j3=51.200, j4=-4.446, j5=73.260, j6=-12.096}
  [445] = {j1=-10.811, j2=60.449, j3=51.735, j4=-4.392, j5=72.819, j6=-12.562}
  [446] = {j1=-10.834, j2=59.913, j3=52.255, j4=-4.341, j5=72.406, j6=-13.009}
  [447] = {j1=-10.856, j2=59.392, j3=52.748, j4=-4.293, j5=72.035, j6=-13.426}
  [448] = {j1=-10.878, j2=58.891, j3=53.203, j4=-4.251, j5=71.720, j6=-13.804}
  [449] = {j1=-10.894, j2=58.474, j3=53.564, j4=-4.220, j5=71.499, j6=-14.097}
  [450] = {j1=-10.910, j2=58.072, j3=53.898, j4=-4.192, j5=71.316, j6=-14.362}
  [451] = {j1=-10.926, j2=57.679, j3=54.216, j4=-4.168, j5=71.159, j6=-14.610}
  [452] = {j1=-10.941, j2=57.288, j3=54.528, j4=-4.144, j5=71.010, j6=-14.852}
  [453] = {j1=-10.941, j2=57.274, j3=54.539, j4=-4.143, j5=71.004, j6=-14.861}
  [454] = {j1=-10.943, j2=57.315, j3=54.465, j4=-4.135, j5=71.118, j6=-14.794}
  [455] = {j1=-10.943, j2=57.330, j3=54.453, j4=-4.136, j5=71.124, j6=-14.785}
  [456] = {j1=-10.927, j2=57.722, j3=54.138, j4=-4.160, j5=71.277, j6=-14.540}
  [457] = {j1=-10.912, j2=58.118, j3=53.817, j4=-4.184, j5=71.440, j6=-14.289}
  [458] = {j1=-10.896, j2=58.521, j3=53.479, j4=-4.211, j5=71.627, j6=-14.022}
  [459] = {j1=-10.879, j2=58.939, j3=53.116, j4=-4.242, j5=71.851, j6=-13.728}
  [460] = {j1=-10.858, j2=59.439, j3=52.662, j4=-4.283, j5=72.165, j6=-13.351}
  [461] = {j1=-10.836, j2=59.959, j3=52.172, j4=-4.331, j5=72.534, j6=-12.936}
  [462] = {j1=-10.813, j2=60.493, j3=51.656, j4=-4.382, j5=72.942, j6=-12.492}
  [463] = {j1=-10.790, j2=61.036, j3=51.125, j4=-4.436, j5=73.378, j6=-12.029}
  [464] = {j1=-10.768, j2=61.581, j3=50.587, j4=-4.489, j5=73.828, j6=-11.556}
  [465] = {j1=-10.747, j2=62.125, j3=50.053, j4=-4.540, j5=74.280, j6=-11.084}
  [466] = {j1=-10.728, j2=62.661, j3=49.530, j4=-4.587, j5=74.721, j6=-10.621}
  [467] = {j1=-10.725, j2=62.754, j3=49.441, j4=-4.594, j5=74.796, j6=-10.542}
  [468] = {j1=-10.710, j2=63.268, j3=48.954, j4=-4.632, j5=75.197, j6=-10.110}
  [469] = {j1=-10.697, j2=63.827, j3=48.463, j4=-4.665, j5=75.567, j6=-9.669}
  [470] = {j1=-10.689, j2=64.310, j3=48.112, j4=-4.688, j5=75.760, j6=-9.340}
  [471] = {j1=-10.683, j2=64.633, j3=47.956, j4=-4.712, j5=75.745, j6=-9.169}
  [472] = {j1=-10.674, j2=64.897, j3=47.910, j4=-4.754, j5=75.584, j6=-9.076}
  [473] = {j1=-10.662, j2=65.108, j3=47.957, j4=-4.816, j5=75.297, j6=-9.048}
  [474] = {j1=-10.646, j2=65.275, j3=48.080, j4=-4.898, j5=74.903, j6=-9.076}
  [475] = {j1=-10.626, j2=65.407, j3=48.263, j4=-5.003, j5=74.421, j6=-9.146}
  [476] = {j1=-10.600, j2=65.509, j3=48.492, j4=-5.136, j5=73.869, j6=-9.246}
  [477] = {j1=-10.569, j2=65.589, j3=48.754, j4=-5.301, j5=73.266, j6=-9.362}
  [478] = {j1=-10.568, j2=65.606, j3=48.724, j4=-5.307, j5=73.325, j6=-9.318}
  [479] = {j1=-10.599, j2=65.527, j3=48.461, j4=-5.141, j5=73.929, j6=-9.201}
  [480] = {j1=-10.625, j2=65.426, j3=48.230, j4=-5.008, j5=74.482, j6=-9.101}
  [481] = {j1=-10.645, j2=65.295, j3=48.045, j4=-4.901, j5=74.965, j6=-9.032}
  [482] = {j1=-10.661, j2=65.128, j3=47.921, j4=-4.818, j5=75.360, j6=-9.005}
  [483] = {j1=-10.674, j2=64.918, j3=47.873, j4=-4.755, j5=75.648, j6=-9.034}
  [484] = {j1=-10.683, j2=64.655, j3=47.918, j4=-4.712, j5=75.809, j6=-9.128}
  [485] = {j1=-10.689, j2=64.331, j3=48.074, j4=-4.686, j5=75.824, j6=-9.301}
  [486] = {j1=-10.698, j2=63.848, j3=48.426, j4=-4.661, j5=75.631, j6=-9.632}
  [487] = {j1=-10.712, j2=63.289, j3=48.917, j4=-4.626, j5=75.260, j6=-10.075}
  [488] = {j1=-10.727, j2=62.775, j3=49.403, j4=-4.589, j5=74.859, j6=-10.508}
  [489] = {j1=-10.730, j2=62.683, j3=49.492, j4=-4.581, j5=74.785, j6=-10.587}
  [490] = {j1=-10.748, j2=62.147, j3=50.013, j4=-4.535, j5=74.346, j6=-11.049}
  [491] = {j1=-10.769, j2=61.605, j3=50.544, j4=-4.484, j5=73.897, j6=-11.520}
  [492] = {j1=-10.791, j2=61.061, j3=51.079, j4=-4.430, j5=73.450, j6=-11.991}
  [493] = {j1=-10.814, j2=60.521, j3=51.607, j4=-4.377, j5=73.018, j6=-12.452}
  [494] = {j1=-10.837, j2=59.989, j3=52.119, j4=-4.326, j5=72.613, j6=-12.894}
  [495] = {j1=-10.859, j2=59.470, j3=52.607, j4=-4.279, j5=72.247, j6=-13.308}
  [496] = {j1=-10.880, j2=58.970, j3=53.061, j4=-4.238, j5=71.933, j6=-13.685}
  [497] = {j1=-10.897, j2=58.552, j3=53.424, j4=-4.207, j5=71.708, j6=-13.980}
  [498] = {j1=-10.913, j2=58.148, j3=53.763, j4=-4.181, j5=71.520, j6=-14.249}
  [499] = {j1=-10.928, j2=57.751, j3=54.086, j4=-4.156, j5=71.354, j6=-14.502}
  [500] = {j1=-10.943, j2=57.358, j3=54.403, j4=-4.132, j5=71.198, j6=-14.748}
  [501] = {j1=-10.944, j2=57.344, j3=54.414, j4=-4.132, j5=71.193, j6=-14.757}
  [502] = {j1=-10.945, j2=57.366, j3=54.374, j4=-4.127, j5=71.254, j6=-14.721}
  [503] = {j1=-10.944, j2=57.381, j3=54.362, j4=-4.128, j5=71.260, j6=-14.712}
  [504] = {j1=-10.929, j2=57.775, j3=54.043, j4=-4.152, j5=71.420, j6=-14.464}
  [505] = {j1=-10.914, j2=58.173, j3=53.717, j4=-4.176, j5=71.589, j6=-14.209}
  [506] = {j1=-10.898, j2=58.579, j3=53.376, j4=-4.202, j5=71.781, j6=-13.938}
  [507] = {j1=-10.881, j2=58.998, j3=53.011, j4=-4.233, j5=72.008, j6=-13.642}
  [508] = {j1=-10.860, j2=59.498, j3=52.557, j4=-4.274, j5=72.323, j6=-13.265}
  [509] = {j1=-10.838, j2=60.016, j3=52.070, j4=-4.321, j5=72.688, j6=-12.852}
  [510] = {j1=-10.815, j2=60.547, j3=51.560, j4=-4.372, j5=73.091, j6=-12.412}
  [511] = {j1=-10.793, j2=61.086, j3=51.034, j4=-4.425, j5=73.520, j6=-11.952}
  [512] = {j1=-10.770, j2=61.629, j3=50.502, j4=-4.478, j5=73.963, j6=-11.484}
  [513] = {j1=-10.750, j2=62.170, j3=49.973, j4=-4.529, j5=74.410, j6=-11.014}
  [514] = {j1=-10.731, j2=62.705, j3=49.453, j4=-4.576, j5=74.848, j6=-10.552}
  [515] = {j1=-10.728, j2=62.797, j3=49.364, j4=-4.583, j5=74.923, j6=-10.473}
  [516] = {j1=-10.713, j2=63.311, j3=48.877, j4=-4.621, j5=75.325, j6=-10.040}
  [517] = {j1=-10.699, j2=63.871, j3=48.385, j4=-4.657, j5=75.697, j6=-9.596}
  [518] = {j1=-10.690, j2=64.355, j3=48.032, j4=-4.684, j5=75.893, j6=-9.261}
  [519] = {j1=-10.683, j2=64.679, j3=47.876, j4=-4.712, j5=75.879, j6=-9.087}
  [520] = {j1=-10.674, j2=64.941, j3=47.831, j4=-4.757, j5=75.719, j6=-8.991}
  [521] = {j1=-10.661, j2=65.152, j3=47.879, j4=-4.821, j5=75.431, j6=-8.962}
  [522] = {j1=-10.644, j2=65.318, j3=48.005, j4=-4.905, j5=75.036, j6=-8.988}
  [523] = {j1=-10.624, j2=65.448, j3=48.191, j4=-5.013, j5=74.552, j6=-9.057}
  [524] = {j1=-10.598, j2=65.549, j3=48.422, j4=-5.147, j5=73.999, j6=-9.157}
  [525] = {j1=-10.567, j2=65.628, j3=48.686, j4=-5.313, j5=73.395, j6=-9.273}
  [526] = {j1=-10.565, j2=65.650, j3=48.647, j4=-5.321, j5=73.473, j6=-9.214}
  [527] = {j1=-10.597, j2=65.573, j3=48.381, j4=-5.154, j5=74.078, j6=-9.098}
  [528] = {j1=-10.623, j2=65.473, j3=48.148, j4=-5.018, j5=74.633, j6=-8.998}
  [529] = {j1=-10.644, j2=65.344, j3=47.960, j4=-4.909, j5=75.118, j6=-8.930}
  [530] = {j1=-10.660, j2=65.178, j3=47.833, j4=-4.823, j5=75.514, j6=-8.905}
  [531] = {j1=-10.674, j2=64.969, j3=47.783, j4=-4.758, j5=75.803, j6=-8.935}
  [532] = {j1=-10.684, j2=64.707, j3=47.827, j4=-4.711, j5=75.964, j6=-9.033}
  [533] = {j1=-10.691, j2=64.383, j3=47.983, j4=-4.681, j5=75.976, j6=-9.209}
  [534] = {j1=-10.701, j2=63.899, j3=48.336, j4=-4.652, j5=75.780, j6=-9.546}
  [535] = {j1=-10.715, j2=63.339, j3=48.829, j4=-4.614, j5=75.406, j6=-9.994}
  [536] = {j1=-10.730, j2=62.825, j3=49.315, j4=-4.575, j5=75.004, j6=-10.428}
  [537] = {j1=-10.733, j2=62.733, j3=49.404, j4=-4.568, j5=74.930, j6=-10.506}
  [538] = {j1=-10.752, j2=62.199, j3=49.921, j4=-4.522, j5=74.495, j6=-10.967}
  [539] = {j1=-10.772, j2=61.660, j3=50.447, j4=-4.471, j5=74.052, j6=-11.435}
  [540] = {j1=-10.794, j2=61.120, j3=50.974, j4=-4.418, j5=73.614, j6=-11.901}
  [541] = {j1=-10.817, j2=60.583, j3=51.495, j4=-4.365, j5=73.189, j6=-12.358}
  [542] = {j1=-10.840, j2=60.054, j3=52.002, j4=-4.314, j5=72.791, j6=-12.796}
  [543] = {j1=-10.862, j2=59.537, j3=52.486, j4=-4.267, j5=72.429, j6=-13.208}
  [544] = {j1=-10.882, j2=59.038, j3=52.939, j4=-4.227, j5=72.114, j6=-13.585}
  [545] = {j1=-10.899, j2=58.618, j3=53.306, j4=-4.197, j5=71.885, j6=-13.883}
  [546] = {j1=-10.915, j2=58.211, j3=53.649, j4=-4.171, j5=71.689, j6=-14.156}
  [547] = {j1=-10.930, j2=57.811, j3=53.978, j4=-4.147, j5=71.515, j6=-14.413}
  [548] = {j1=-10.945, j2=57.415, j3=54.300, j4=-4.123, j5=71.352, j6=-14.664}
  [549] = {j1=-10.946, j2=57.401, j3=54.312, j4=-4.122, j5=71.347, j6=-14.673}
  [550] = {j1=-10.947, j2=57.430, j3=54.261, j4=-4.116, j5=71.426, j6=-14.627}
  [551] = {j1=-10.947, j2=57.444, j3=54.249, j4=-4.117, j5=71.432, j6=-14.618}
  [552] = {j1=-10.931, j2=57.842, j3=53.923, j4=-4.140, j5=71.600, j6=-14.364}
  [553] = {j1=-10.916, j2=58.244, j3=53.590, j4=-4.164, j5=71.779, j6=-14.103}
  [554] = {j1=-10.900, j2=58.653, j3=53.243, j4=-4.190, j5=71.980, j6=-13.828}
  [555] = {j1=-10.884, j2=59.075, j3=52.874, j4=-4.220, j5=72.213, j6=-13.528}
  [556] = {j1=-10.863, j2=59.574, j3=52.420, j4=-4.261, j5=72.528, j6=-13.151}
  [557] = {j1=-10.841, j2=60.090, j3=51.938, j4=-4.307, j5=72.889, j6=-12.740}
  [558] = {j1=-10.819, j2=60.618, j3=51.434, j4=-4.357, j5=73.285, j6=-12.304}
  [559] = {j1=-10.796, j2=61.153, j3=50.916, j4=-4.410, j5=73.705, j6=-11.850}
  [560] = {j1=-10.774, j2=61.691, j3=50.392, j4=-4.463, j5=74.139, j6=-11.386}
  [561] = {j1=-10.754, j2=62.228, j3=49.869, j4=-4.514, j5=74.579, j6=-10.920}
  [562] = {j1=-10.735, j2=62.761, j3=49.354, j4=-4.560, j5=75.013, j6=-10.461}
  [563] = {j1=-10.732, j2=62.853, j3=49.265, j4=-4.568, j5=75.087, j6=-10.382}
  [564] = {j1=-10.717, j2=63.367, j3=48.779, j4=-4.607, j5=75.489, j6=-9.947}
  [565] = {j1=-10.702, j2=63.928, j3=48.285, j4=-4.646, j5=75.866, j6=-9.497}
  [566] = {j1=-10.692, j2=64.413, j3=47.930, j4=-4.679, j5=76.064, j6=-9.157}
  [567] = {j1=-10.684, j2=64.737, j3=47.774, j4=-4.710, j5=76.053, j6=-8.979}
  [568] = {j1=-10.673, j2=64.999, j3=47.730, j4=-4.760, j5=75.893, j6=-8.879}
  [569] = {j1=-10.660, j2=65.208, j3=47.781, j4=-4.827, j5=75.604, j6=-8.848}
  [570] = {j1=-10.643, j2=65.373, j3=47.909, j4=-4.914, j5=75.207, j6=-8.872}
  [571] = {j1=-10.622, j2=65.501, j3=48.098, j4=-5.025, j5=74.722, j6=-8.940}
  [572] = {j1=-10.596, j2=65.600, j3=48.333, j4=-5.162, j5=74.167, j6=-9.039}
  [573] = {j1=-10.564, j2=65.677, j3=48.600, j4=-5.330, j5=73.561, j6=-9.154}
  [574] = {j1=-10.562, j2=65.700, j3=48.561, j4=-5.338, j5=73.638, j6=-9.095}
  [575] = {j1=-10.595, j2=65.624, j3=48.293, j4=-5.168, j5=74.245, j6=-8.980}
  [576] = {j1=-10.621, j2=65.525, j3=48.056, j4=-5.030, j5=74.802, j6=-8.882}
  [577] = {j1=-10.642, j2=65.398, j3=47.865, j4=-4.919, j5=75.288, j6=-8.814}
  [578] = {j1=-10.660, j2=65.234, j3=47.735, j4=-4.830, j5=75.686, j6=-8.791}
  [579] = {j1=-10.673, j2=65.026, j3=47.683, j4=-4.761, j5=75.976, j6=-8.823}
  [580] = {j1=-10.684, j2=64.764, j3=47.726, j4=-4.710, j5=76.136, j6=-8.924}
  [581] = {j1=-10.693, j2=64.441, j3=47.881, j4=-4.675, j5=76.148, j6=-9.105}
  [582] = {j1=-10.704, j2=63.956, j3=48.236, j4=-4.641, j5=75.948, j6=-9.448}
  [583] = {j1=-10.719, j2=63.394, j3=48.730, j4=-4.600, j5=75.570, j6=-9.900}
  [584] = {j1=-10.734, j2=62.881, j3=49.216, j4=-4.560, j5=75.168, j6=-10.336}
  [585] = {j1=-10.737, j2=62.789, j3=49.304, j4=-4.553, j5=75.095, j6=-10.414}
  [586] = {j1=-10.756, j2=62.258, j3=49.817, j4=-4.506, j5=74.663, j6=-10.873}
  [587] = {j1=-10.776, j2=61.722, j3=50.337, j4=-4.456, j5=74.228, j6=-11.337}
  [588] = {j1=-10.798, j2=61.186, j3=50.856, j4=-4.403, j5=73.799, j6=-11.798}
  [589] = {j1=-10.820, j2=60.654, j3=51.369, j4=-4.350, j5=73.383, j6=-12.249}
  [590] = {j1=-10.843, j2=60.128, j3=51.870, j4=-4.300, j5=72.992, j6=-12.684}
  [591] = {j1=-10.864, j2=59.613, j3=52.350, j4=-4.254, j5=72.633, j6=-13.094}
  [592] = {j1=-10.885, j2=59.114, j3=52.804, j4=-4.214, j5=72.318, j6=-13.472}
  [593] = {j1=-10.901, j2=58.691, j3=53.174, j4=-4.184, j5=72.082, j6=-13.773}
  [594] = {j1=-10.917, j2=58.280, j3=53.525, j4=-4.159, j5=71.876, j6=-14.052}
  [595] = {j1=-10.932, j2=57.877, j3=53.861, j4=-4.135, j5=71.692, j6=-14.316}
  [596] = {j1=-10.948, j2=57.477, j3=54.190, j4=-4.112, j5=71.520, j6=-14.572}
  [597] = {j1=-10.948, j2=57.463, j3=54.201, j4=-4.111, j5=71.514, j6=-14.581}
  [598] = {j1=-10.950, j2=57.490, j3=54.153, j4=-4.105, j5=71.590, j6=-14.537}
  [599] = {j1=-10.949, j2=57.504, j3=54.141, j4=-4.106, j5=71.597, j6=-14.527}
  [600] = {j1=-10.934, j2=57.906, j3=53.808, j4=-4.129, j5=71.774, j6=-14.268}
  [601] = {j1=-10.918, j2=58.312, j3=53.467, j4=-4.152, j5=71.964, j6=-14.001}
  [602] = {j1=-10.903, j2=58.726, j3=53.113, j4=-4.178, j5=72.175, j6=-13.719}
  [603] = {j1=-10.886, j2=59.150, j3=52.739, j4=-4.207, j5=72.415, j6=-13.415}
  [604] = {j1=-10.866, j2=59.650, j3=52.284, j4=-4.247, j5=72.733, j6=-13.036}
  [605] = {j1=-10.844, j2=60.164, j3=51.805, j4=-4.293, j5=73.090, j6=-12.627}
  [606] = {j1=-10.822, j2=60.688, j3=51.307, j4=-4.343, j5=73.479, j6=-12.195}
  [607] = {j1=-10.800, j2=61.219, j3=50.798, j4=-4.396, j5=73.890, j6=-11.746}
  [608] = {j1=-10.778, j2=61.753, j3=50.282, j4=-4.448, j5=74.316, j6=-11.287}
  [609] = {j1=-10.758, j2=62.287, j3=49.765, j4=-4.499, j5=74.747, j6=-10.826}
  [610] = {j1=-10.739, j2=62.817, j3=49.254, j4=-4.545, j5=75.177, j6=-10.368}
  [611] = {j1=-10.736, j2=62.909, j3=49.166, j4=-4.553, j5=75.251, j6=-10.289}
  [612] = {j1=-10.721, j2=63.423, j3=48.680, j4=-4.593, j5=75.653, j6=-9.854}
  [613] = {j1=-10.705, j2=63.985, j3=48.185, j4=-4.635, j5=76.033, j6=-9.399}
  [614] = {j1=-10.693, j2=64.470, j3=47.829, j4=-4.673, j5=76.235, j6=-9.053}
  [615] = {j1=-10.684, j2=64.794, j3=47.674, j4=-4.709, j5=76.225, j6=-8.870}
  [616] = {j1=-10.673, j2=65.056, j3=47.631, j4=-4.762, j5=76.065, j6=-8.768}
  [617] = {j1=-10.659, j2=65.264, j3=47.684, j4=-4.833, j5=75.775, j6=-8.734}
  [618] = {j1=-10.641, j2=65.427, j3=47.815, j4=-4.924, j5=75.377, j6=-8.757}
  [619] = {j1=-10.620, j2=65.553, j3=48.007, j4=-5.037, j5=74.890, j6=-8.824}
  [620] = {j1=-10.593, j2=65.651, j3=48.246, j4=-5.176, j5=74.333, j6=-8.922}
  [621] = {j1=-10.561, j2=65.726, j3=48.515, j4=-5.346, j5=73.725, j6=-9.037}
  [622] = {j1=-10.559, j2=65.748, j3=48.477, j4=-5.354, j5=73.802, j6=-8.978}
  [623] = {j1=-10.592, j2=65.674, j3=48.206, j4=-5.183, j5=74.410, j6=-8.864}
  [624] = {j1=-10.619, j2=65.577, j3=47.966, j4=-5.042, j5=74.968, j6=-8.766}
  [625] = {j1=-10.641, j2=65.452, j3=47.771, j4=-4.928, j5=75.457, j6=-8.700}
  [626] = {j1=-10.659, j2=65.290, j3=47.639, j4=-4.836, j5=75.856, j6=-8.677}
  [627] = {j1=-10.673, j2=65.082, j3=47.584, j4=-4.763, j5=76.147, j6=-8.712}
  [628] = {j1=-10.685, j2=64.821, j3=47.626, j4=-4.708, j5=76.307, j6=-8.816}
  [629] = {j1=-10.694, j2=64.498, j3=47.781, j4=-4.669, j5=76.318, j6=-9.001}
  [630] = {j1=-10.707, j2=64.012, j3=48.137, j4=-4.629, j5=76.114, j6=-9.350}
  [631] = {j1=-10.723, j2=63.450, j3=48.632, j4=-4.586, j5=75.734, j6=-9.807}
  [632] = {j1=-10.738, j2=62.937, j3=49.117, j4=-4.545, j5=75.332, j6=-10.243}
  [633] = {j1=-10.741, j2=62.845, j3=49.204, j4=-4.537, j5=75.259, j6=-10.322}
  [634] = {j1=-10.760, j2=62.316, j3=49.713, j4=-4.491, j5=74.832, j6=-10.778}
  [635] = {j1=-10.780, j2=61.785, j3=50.226, j4=-4.441, j5=74.405, j6=-11.237}
  [636] = {j1=-10.801, j2=61.253, j3=50.737, j4=-4.389, j5=73.984, j6=-11.693}
  [637] = {j1=-10.823, j2=60.725, j3=51.243, j4=-4.336, j5=73.578, j6=-12.140}
  [638] = {j1=-10.846, j2=60.202, j3=51.737, j4=-4.287, j5=73.193, j6=-12.571}
  [639] = {j1=-10.867, j2=59.689, j3=52.215, j4=-4.241, j5=72.837, j6=-12.979}
  [640] = {j1=-10.887, j2=59.189, j3=52.669, j4=-4.201, j5=72.519, j6=-13.359}
  [641] = {j1=-10.904, j2=58.763, j3=53.046, j4=-4.172, j5=72.275, j6=-13.665}
  [642] = {j1=-10.920, j2=58.347, j3=53.404, j4=-4.147, j5=72.058, j6=-13.950}
  [643] = {j1=-10.935, j2=57.939, j3=53.749, j4=-4.123, j5=71.863, j6=-14.221}
  [644] = {j1=-10.950, j2=57.536, j3=54.085, j4=-4.100, j5=71.681, j6=-14.483}
  [645] = {j1=-10.951, j2=57.521, j3=54.097, j4=-4.100, j5=71.675, j6=-14.493}
  [646] = {j1=-10.952, j2=57.547, j3=54.051, j4=-4.093, j5=71.748, j6=-14.450}
  [647] = {j1=-10.952, j2=57.562, j3=54.038, j4=-4.094, j5=71.754, j6=-14.440}
  [648] = {j1=-10.936, j2=57.967, j3=53.698, j4=-4.117, j5=71.941, j6=-14.175}
  [649] = {j1=-10.921, j2=58.379, j3=53.348, j4=-4.140, j5=72.144, j6=-13.901}
  [650] = {j1=-10.905, j2=58.797, j3=52.985, j4=-4.165, j5=72.367, j6=-13.612}
  [651] = {j1=-10.889, j2=59.225, j3=52.605, j4=-4.194, j5=72.615, j6=-13.303}
  [652] = {j1=-10.869, j2=59.726, j3=52.149, j4=-4.234, j5=72.936, j6=-12.922}
  [653] = {j1=-10.847, j2=60.238, j3=51.672, j4=-4.280, j5=73.291, j6=-12.514}
  [654] = {j1=-10.825, j2=60.759, j3=51.181, j4=-4.329, j5=73.673, j6=-12.085}
  [655] = {j1=-10.803, j2=61.286, j3=50.678, j4=-4.381, j5=74.076, j6=-11.641}
  [656] = {j1=-10.782, j2=61.816, j3=50.170, j4=-4.434, j5=74.493, j6=-11.187}
  [657] = {j1=-10.762, j2=62.346, j3=49.661, j4=-4.484, j5=74.917, j6=-10.730}
  [658] = {j1=-10.743, j2=62.874, j3=49.154, j4=-4.530, j5=75.341, j6=-10.275}
  [659] = {j1=-10.740, j2=62.965, j3=49.066, j4=-4.537, j5=75.415, j6=-10.196}
  [660] = {j1=-10.724, j2=63.478, j3=48.582, j4=-4.579, j5=75.817, j6=-9.760}
  [661] = {j1=-10.708, j2=64.041, j3=48.086, j4=-4.624, j5=76.199, j6=-9.301}
  [662] = {j1=-10.695, j2=64.527, j3=47.729, j4=-4.666, j5=76.404, j6=-8.949}
  [663] = {j1=-10.685, j2=64.851, j3=47.574, j4=-4.708, j5=76.395, j6=-8.763}
  [664] = {j1=-10.673, j2=65.111, j3=47.533, j4=-4.765, j5=76.234, j6=-8.657}
  [665] = {j1=-10.658, j2=65.318, j3=47.589, j4=-4.839, j5=75.944, j6=-8.621}
  [666] = {j1=-10.640, j2=65.480, j3=47.723, j4=-4.933, j5=75.544, j6=-8.643}
  [667] = {j1=-10.618, j2=65.604, j3=47.918, j4=-5.049, j5=75.055, j6=-8.709}
  [668] = {j1=-10.591, j2=65.700, j3=48.159, j4=-5.190, j5=74.496, j6=-8.806}
  [669] = {j1=-10.558, j2=65.774, j3=48.432, j4=-5.363, j5=73.887, j6=-8.920}
  [670] = {j1=-10.557, j2=65.796, j3=48.394, j4=-5.370, j5=73.963, j6=-8.862}
  [671] = {j1=-10.589, j2=65.723, j3=48.120, j4=-5.197, j5=74.573, j6=-8.748}
  [672] = {j1=-10.617, j2=65.628, j3=47.877, j4=-5.054, j5=75.133, j6=-8.651}
  [673] = {j1=-10.639, j2=65.504, j3=47.680, j4=-4.937, j5=75.623, j6=-8.586}
  [674] = {j1=-10.658, j2=65.344, j3=47.544, j4=-4.842, j5=76.024, j6=-8.565}
  [675] = {j1=-10.673, j2=65.138, j3=47.487, j4=-4.766, j5=76.316, j6=-8.602}
  [676] = {j1=-10.686, j2=64.878, j3=47.527, j4=-4.707, j5=76.477, j6=-8.709}
  [677] = {j1=-10.696, j2=64.555, j3=47.681, j4=-4.663, j5=76.486, j6=-8.898}
  [678] = {j1=-10.710, j2=64.068, j3=48.038, j4=-4.618, j5=76.280, j6=-9.252}
  [679] = {j1=-10.726, j2=63.506, j3=48.534, j4=-4.571, j5=75.898, j6=-9.712}
  [680] = {j1=-10.742, j2=62.993, j3=49.017, j4=-4.530, j5=75.497, j6=-10.150}
  [681] = {j1=-10.745, j2=62.902, j3=49.104, j4=-4.522, j5=75.424, j6=-10.228}
  [682] = {j1=-10.763, j2=62.375, j3=49.608, j4=-4.476, j5=75.002, j6=-10.682}
  [683] = {j1=-10.783, j2=61.847, j3=50.114, j4=-4.426, j5=74.582, j6=-11.137}
  [684] = {j1=-10.805, j2=61.320, j3=50.618, j4=-4.374, j5=74.170, j6=-11.588}
  [685] = {j1=-10.827, j2=60.796, j3=51.116, j4=-4.323, j5=73.772, j6=-12.030}
  [686] = {j1=-10.848, j2=60.276, j3=51.605, j4=-4.273, j5=73.393, j6=-12.457}
  [687] = {j1=-10.870, j2=59.765, j3=52.080, j4=-4.228, j5=73.040, j6=-12.864}
  [688] = {j1=-10.890, j2=59.263, j3=52.537, j4=-4.188, j5=72.717, j6=-13.247}
  [689] = {j1=-10.907, j2=58.834, j3=52.920, j4=-4.159, j5=72.464, j6=-13.559}
  [690] = {j1=-10.922, j2=58.413, j3=53.288, j4=-4.134, j5=72.235, j6=-13.852}
  [691] = {j1=-10.938, j2=57.999, j3=53.642, j4=-4.111, j5=72.027, j6=-14.130}
  [692] = {j1=-10.953, j2=57.591, j3=53.986, j4=-4.089, j5=71.835, j6=-14.398}
  [693] = {j1=-10.954, j2=57.576, j3=53.998, j4=-4.088, j5=71.829, j6=-14.408}
  [694] = {j1=-10.955, j2=57.601, j3=53.954, j4=-4.082, j5=71.898, j6=-14.367}
  [695] = {j1=-10.955, j2=57.616, j3=53.942, j4=-4.082, j5=71.905, j6=-14.357}
  [696] = {j1=-10.939, j2=58.026, j3=53.594, j4=-4.105, j5=72.103, j6=-14.086}
  [697] = {j1=-10.924, j2=58.443, j3=53.234, j4=-4.127, j5=72.318, j6=-13.803}
  [698] = {j1=-10.908, j2=58.867, j3=52.861, j4=-4.152, j5=72.554, j6=-13.507}
  [699] = {j1=-10.892, j2=59.298, j3=52.474, j4=-4.181, j5=72.813, j6=-13.192}
  [700] = {j1=-10.871, j2=59.801, j3=52.014, j4=-4.221, j5=73.138, j6=-12.807}
  [701] = {j1=-10.850, j2=60.313, j3=51.540, j4=-4.266, j5=73.492, j6=-12.400}
  [702] = {j1=-10.828, j2=60.831, j3=51.053, j4=-4.316, j5=73.868, j6=-11.974}
  [703] = {j1=-10.806, j2=61.353, j3=50.559, j4=-4.367, j5=74.263, j6=-11.534}
  [704] = {j1=-10.785, j2=61.879, j3=50.058, j4=-4.419, j5=74.671, j6=-11.086}
  [705] = {j1=-10.765, j2=62.405, j3=49.556, j4=-4.469, j5=75.087, j6=-10.633}
  [706] = {j1=-10.747, j2=62.930, j3=49.054, j4=-4.515, j5=75.506, j6=-10.181}
  [707] = {j1=-10.744, j2=63.021, j3=48.967, j4=-4.522, j5=75.579, j6=-10.103}
  [708] = {j1=-10.728, j2=63.534, j3=48.484, j4=-4.564, j5=75.980, j6=-9.665}
  [709] = {j1=-10.711, j2=64.097, j3=47.988, j4=-4.613, j5=76.364, j6=-9.203}
  [710] = {j1=-10.697, j2=64.584, j3=47.631, j4=-4.660, j5=76.571, j6=-8.846}
  [711] = {j1=-10.686, j2=64.907, j3=47.476, j4=-4.706, j5=76.563, j6=-8.655}
  [712] = {j1=-10.673, j2=65.166, j3=47.437, j4=-4.767, j5=76.402, j6=-8.547}
  [713] = {j1=-10.657, j2=65.372, j3=47.495, j4=-4.845, j5=76.110, j6=-8.509}
  [714] = {j1=-10.638, j2=65.532, j3=47.632, j4=-4.942, j5=75.708, j6=-8.529}
  [715] = {j1=-10.616, j2=65.655, j3=47.831, j4=-5.061, j5=75.217, j6=-8.594}
  [716] = {j1=-10.588, j2=65.749, j3=48.075, j4=-5.205, j5=74.657, j6=-8.690}
  [717] = {j1=-10.555, j2=65.821, j3=48.350, j4=-5.379, j5=74.047, j6=-8.804}
  [718] = {j1=-10.554, j2=65.843, j3=48.313, j4=-5.387, j5=74.122, j6=-8.746}
  [719] = {j1=-10.587, j2=65.771, j3=48.036, j4=-5.211, j5=74.733, j6=-8.633}
  [720] = {j1=-10.615, j2=65.678, j3=47.790, j4=-5.066, j5=75.295, j6=-8.537}
  [721] = {j1=-10.638, j2=65.556, j3=47.590, j4=-4.946, j5=75.787, j6=-8.473}
  [722] = {j1=-10.657, j2=65.397, j3=47.451, j4=-4.848, j5=76.189, j6=-8.454}
  [723] = {j1=-10.673, j2=65.193, j3=47.392, j4=-4.768, j5=76.482, j6=-8.492}
  [724] = {j1=-10.686, j2=64.934, j3=47.429, j4=-4.705, j5=76.644, j6=-8.602}
  [725] = {j1=-10.698, j2=64.611, j3=47.583, j4=-4.657, j5=76.653, j6=-8.795}
  [726] = {j1=-10.713, j2=64.124, j3=47.940, j4=-4.607, j5=76.445, j6=-9.154}
  [727] = {j1=-10.730, j2=63.561, j3=48.436, j4=-4.557, j5=76.061, j6=-9.618}
  [728] = {j1=-10.746, j2=63.049, j3=48.917, j4=-4.515, j5=75.661, j6=-10.055}
  [729] = {j1=-10.749, j2=62.959, j3=49.004, j4=-4.507, j5=75.588, j6=-10.134}
  [730] = {j1=-10.767, j2=62.435, j3=49.503, j4=-4.462, j5=75.172, j6=-10.584}
  [731] = {j1=-10.787, j2=61.911, j3=50.002, j4=-4.412, j5=74.760, j6=-11.035}
  [732] = {j1=-10.808, j2=61.388, j3=50.498, j4=-4.361, j5=74.357, j6=-11.481}
  [733] = {j1=-10.830, j2=60.867, j3=50.989, j4=-4.309, j5=73.967, j6=-11.918}
  [734] = {j1=-10.851, j2=60.351, j3=51.472, j4=-4.260, j5=73.594, j6=-12.342}
  [735] = {j1=-10.873, j2=59.840, j3=51.946, j4=-4.214, j5=73.241, j6=-12.750}
  [736] = {j1=-10.893, j2=59.336, j3=52.406, j4=-4.175, j5=72.913, j6=-13.136}
  [737] = {j1=-10.910, j2=58.902, j3=52.797, j4=-4.146, j5=72.649, j6=-13.455}
  [738] = {j1=-10.925, j2=58.476, j3=53.175, j4=-4.121, j5=72.407, j6=-13.756}
  [739] = {j1=-10.941, j2=58.056, j3=53.540, j4=-4.099, j5=72.184, j6=-14.042}
  [740] = {j1=-10.956, j2=57.643, j3=53.892, j4=-4.077, j5=71.982, j6=-14.317}
  [741] = {j1=-10.957, j2=57.629, j3=53.905, j4=-4.076, j5=71.975, j6=-14.327}
  [742] = {j1=-10.958, j2=57.652, j3=53.864, j4=-4.069, j5=72.041, j6=-14.288}
  [743] = {j1=-10.958, j2=57.667, j3=53.851, j4=-4.070, j5=72.048, j6=-14.278}
  [744] = {j1=-10.943, j2=58.082, j3=53.494, j4=-4.092, j5=72.257, j6=-14.000}
  [745] = {j1=-10.927, j2=58.505, j3=53.123, j4=-4.114, j5=72.488, j6=-13.709}
  [746] = {j1=-10.911, j2=58.935, j3=52.739, j4=-4.138, j5=72.738, j6=-13.403}
  [747] = {j1=-10.895, j2=59.371, j3=52.344, j4=-4.167, j5=73.008, j6=-13.081}
  [748] = {j1=-10.874, j2=59.876, j3=51.881, j4=-4.207, j5=73.339, j6=-12.693}
  [749] = {j1=-10.853, j2=60.387, j3=51.407, j4=-4.253, j5=73.692, j6=-12.285}
  [750] = {j1=-10.831, j2=60.902, j3=50.926, j4=-4.302, j5=74.064, j6=-11.862}
  [751] = {j1=-10.810, j2=61.421, j3=50.438, j4=-4.354, j5=74.450, j6=-11.427}
  [752] = {j1=-10.789, j2=61.942, j3=49.946, j4=-4.405, j5=74.849, j6=-10.983}
  [753] = {j1=-10.769, j2=62.465, j3=49.450, j4=-4.454, j5=75.257, j6=-10.535}
  [754] = {j1=-10.751, j2=62.987, j3=48.954, j4=-4.500, j5=75.671, j6=-10.086}
  [755] = {j1=-10.748, j2=63.078, j3=48.867, j4=-4.507, j5=75.744, j6=-10.008}
  [756] = {j1=-10.732, j2=63.589, j3=48.386, j4=-4.550, j5=76.143, j6=-9.570}
  [757] = {j1=-10.715, j2=64.152, j3=47.890, j4=-4.601, j5=76.528, j6=-9.105}
  [758] = {j1=-10.699, j2=64.639, j3=47.533, j4=-4.654, j5=76.737, j6=-8.743}
  [759] = {j1=-10.687, j2=64.962, j3=47.380, j4=-4.704, j5=76.728, j6=-8.549}
  [760] = {j1=-10.673, j2=65.220, j3=47.343, j4=-4.770, j5=76.567, j6=-8.438}
  [761] = {j1=-10.656, j2=65.424, j3=47.403, j4=-4.851, j5=76.274, j6=-8.398}
  [762] = {j1=-10.637, j2=65.583, j3=47.543, j4=-4.951, j5=75.870, j6=-8.417}
  [763] = {j1=-10.613, j2=65.704, j3=47.745, j4=-5.072, j5=75.378, j6=-8.481}
  [764] = {j1=-10.586, j2=65.796, j3=47.992, j4=-5.219, j5=74.816, j6=-8.576}
  [765] = {j1=-10.552, j2=65.867, j3=48.270, j4=-5.395, j5=74.205, j6=-8.688}
  [766] = {j1=-10.551, j2=65.889, j3=48.233, j4=-5.403, j5=74.279, j6=-8.631}
  [767] = {j1=-10.585, j2=65.819, j3=47.953, j4=-5.226, j5=74.891, j6=-8.519}
  [768] = {j1=-10.613, j2=65.727, j3=47.705, j4=-5.078, j5=75.454, j6=-8.424}
  [769] = {j1=-10.636, j2=65.607, j3=47.501, j4=-4.955, j5=75.948, j6=-8.361}
  [770] = {j1=-10.656, j2=65.449, j3=47.360, j4=-4.854, j5=76.352, j6=-8.343}
  [771] = {j1=-10.673, j2=65.246, j3=47.298, j4=-4.771, j5=76.646, j6=-8.384}
  [772] = {j1=-10.687, j2=64.988, j3=47.333, j4=-4.703, j5=76.809, j6=-8.496}
  [773] = {j1=-10.700, j2=64.666, j3=47.486, j4=-4.650, j5=76.818, j6=-8.692}
  [774] = {j1=-10.716, j2=64.179, j3=47.842, j4=-4.595, j5=76.609, j6=-9.056}
  [775] = {j1=-10.734, j2=63.617, j3=48.338, j4=-4.542, j5=76.224, j6=-9.523}
  [776] = {j1=-10.750, j2=63.106, j3=48.817, j4=-4.499, j5=75.826, j6=-9.960}
  [777] = {j1=-10.753, j2=63.015, j3=48.903, j4=-4.492, j5=75.754, j6=-10.038}
  [778] = {j1=-10.771, j2=62.495, j3=49.397, j4=-4.447, j5=75.343, j6=-10.486}
  [779] = {j1=-10.790, j2=61.974, j3=49.888, j4=-4.398, j5=74.939, j6=-10.931}
  [780] = {j1=-10.811, j2=61.456, j3=50.377, j4=-4.347, j5=74.545, j6=-11.372}
  [781] = {j1=-10.833, j2=60.939, j3=50.861, j4=-4.296, j5=74.162, j6=-11.805}
  [782] = {j1=-10.854, j2=60.425, j3=51.340, j4=-4.246, j5=73.794, j6=-12.228}
  [783] = {j1=-10.876, j2=59.914, j3=51.812, j4=-4.201, j5=73.441, j6=-12.636}
  [784] = {j1=-10.896, j2=59.408, j3=52.278, j4=-4.161, j5=73.107, j6=-13.027}
  [785] = {j1=-10.913, j2=58.969, j3=52.677, j4=-4.132, j5=72.831, j6=-13.352}
  [786] = {j1=-10.929, j2=58.536, j3=53.067, j4=-4.107, j5=72.573, j6=-13.663}
  [787] = {j1=-10.944, j2=58.110, j3=53.444, j4=-4.086, j5=72.335, j6=-13.958}
  [788] = {j1=-10.959, j2=57.692, j3=53.805, j4=-4.065, j5=72.121, j6=-14.239}
  [789] = {j1=-10.960, j2=57.678, j3=53.817, j4=-4.064, j5=72.113, j6=-14.249}
  [790] = {j1=-10.962, j2=57.699, j3=53.779, j4=-4.057, j5=72.176, j6=-14.212}
  [791] = {j1=-10.961, j2=57.714, j3=53.766, j4=-4.058, j5=72.184, j6=-14.202}
  [792] = {j1=-10.946, j2=58.134, j3=53.400, j4=-4.079, j5=72.405, j6=-13.917}
  [793] = {j1=-10.931, j2=58.564, j3=53.017, j4=-4.100, j5=72.651, j6=-13.617}
  [794] = {j1=-10.915, j2=59.001, j3=52.620, j4=-4.124, j5=72.918, j6=-13.302}
  [795] = {j1=-10.898, j2=59.443, j3=52.216, j4=-4.154, j5=73.200, j6=-12.972}
  [796] = {j1=-10.877, j2=59.951, j3=51.748, j4=-4.194, j5=73.539, j6=-12.578}
  [797] = {j1=-10.856, j2=60.461, j3=51.275, j4=-4.240, j5=73.892, j6=-12.170}
  [798] = {j1=-10.834, j2=60.974, j3=50.798, j4=-4.289, j5=74.259, j6=-11.749}
  [799] = {j1=-10.813, j2=61.489, j3=50.317, j4=-4.340, j5=74.638, j6=-11.318}
  [800] = {j1=-10.792, j2=62.006, j3=49.832, j4=-4.391, j5=75.028, j6=-10.879}
  [801] = {j1=-10.773, j2=62.525, j3=49.344, j4=-4.440, j5=75.428, j6=-10.436}
  [802] = {j1=-10.755, j2=63.044, j3=48.853, j4=-4.485, j5=75.837, j6=-9.990}
  [803] = {j1=-10.752, j2=63.135, j3=48.767, j4=-4.492, j5=75.908, j6=-9.912}
  [804] = {j1=-10.736, j2=63.645, j3=48.288, j4=-4.535, j5=76.306, j6=-9.475}
  [805] = {j1=-10.718, j2=64.207, j3=47.793, j4=-4.589, j5=76.691, j6=-9.007}
  [806] = {j1=-10.701, j2=64.694, j3=47.437, j4=-4.647, j5=76.901, j6=-8.640}
  [807] = {j1=-10.688, j2=65.016, j3=47.285, j4=-4.703, j5=76.892, j6=-8.443}
  [808] = {j1=-10.673, j2=65.274, j3=47.250, j4=-4.772, j5=76.730, j6=-8.330}
  [809] = {j1=-10.655, j2=65.476, j3=47.313, j4=-4.857, j5=76.435, j6=-8.288}
  [810] = {j1=-10.635, j2=65.633, j3=47.456, j4=-4.960, j5=76.030, j6=-8.305}
  [811] = {j1=-10.611, j2=65.752, j3=47.661, j4=-5.084, j5=75.535, j6=-8.368}
  [812] = {j1=-10.583, j2=65.843, j3=47.911, j4=-5.233, j5=74.972, j6=-8.462}
  [813] = {j1=-10.549, j2=65.913, j3=48.191, j4=-5.411, j5=74.360, j6=-8.574}
  [814] = {j1=-10.548, j2=65.934, j3=48.154, j4=-5.419, j5=74.434, j6=-8.517}
  [815] = {j1=-10.582, j2=65.865, j3=47.873, j4=-5.240, j5=75.046, j6=-8.406}
  [816] = {j1=-10.611, j2=65.775, j3=47.621, j4=-5.090, j5=75.611, j6=-8.312}
  [817] = {j1=-10.635, j2=65.656, j3=47.415, j4=-4.964, j5=76.106, j6=-8.250}
  [818] = {j1=-10.655, j2=65.501, j3=47.270, j4=-4.860, j5=76.512, j6=-8.233}
  [819] = {j1=-10.673, j2=65.299, j3=47.206, j4=-4.773, j5=76.808, j6=-8.276}
  [820] = {j1=-10.688, j2=65.042, j3=47.239, j4=-4.701, j5=76.972, j6=-8.390}
  [821] = {j1=-10.702, j2=64.721, j3=47.390, j4=-4.644, j5=76.981, j6=-8.589}
  [822] = {j1=-10.719, j2=64.234, j3=47.745, j4=-4.584, j5=76.771, j6=-8.958}
  [823] = {j1=-10.738, j2=63.672, j3=48.240, j4=-4.528, j5=76.387, j6=-9.427}
  [824] = {j1=-10.754, j2=63.163, j3=48.717, j4=-4.484, j5=75.991, j6=-9.864}
  [825] = {j1=-10.757, j2=63.073, j3=48.802, j4=-4.477, j5=75.919, j6=-9.941}
  [826] = {j1=-10.775, j2=62.555, j3=49.290, j4=-4.433, j5=75.514, j6=-10.385}
  [827] = {j1=-10.794, j2=62.039, j3=49.774, j4=-4.384, j5=75.119, j6=-10.827}
  [828] = {j1=-10.814, j2=61.524, j3=50.255, j4=-4.333, j5=74.733, j6=-11.263}
  [829] = {j1=-10.836, j2=61.011, j3=50.733, j4=-4.282, j5=74.358, j6=-11.692}
  [830] = {j1=-10.857, j2=60.499, j3=51.208, j4=-4.233, j5=73.993, j6=-12.112}
  [831] = {j1=-10.878, j2=59.988, j3=51.680, j4=-4.187, j5=73.640, j6=-12.521}
  [832] = {j1=-10.899, j2=59.479, j3=52.151, j4=-4.147, j5=73.297, j6=-12.918}
  [833] = {j1=-10.916, j2=59.034, j3=52.561, j4=-4.117, j5=73.008, j6=-13.252}
  [834] = {j1=-10.932, j2=58.594, j3=52.963, j4=-4.093, j5=72.734, j6=-13.572}
  [835] = {j1=-10.948, j2=58.161, j3=53.353, j4=-4.072, j5=72.480, j6=-13.877}
  [836] = {j1=-10.963, j2=57.738, j3=53.723, j4=-4.052, j5=72.252, j6=-14.166}
  [837] = {j1=-10.963, j2=57.723, j3=53.736, j4=-4.051, j5=72.244, j6=-14.176}
  [838] = {j1=-10.965, j2=57.743, j3=53.700, j4=-4.044, j5=72.304, j6=-14.141}
  [839] = {j1=-10.965, j2=57.759, j3=53.687, j4=-4.045, j5=72.312, j6=-14.130}
  [840] = {j1=-10.950, j2=58.184, j3=53.311, j4=-4.065, j5=72.547, j6=-13.838}
  [841] = {j1=-10.934, j2=58.621, j3=52.915, j4=-4.086, j5=72.810, j6=-13.528}
  [842] = {j1=-10.918, j2=59.066, j3=52.505, j4=-4.110, j5=73.093, j6=-13.203}
  [843] = {j1=-10.901, j2=59.513, j3=52.090, j4=-4.139, j5=73.390, j6=-12.864}
  [844] = {j1=-10.880, j2=60.025, j3=51.616, j4=-4.180, j5=73.737, j6=-12.464}
  [845] = {j1=-10.859, j2=60.535, j3=51.142, j4=-4.226, j5=74.092, j6=-12.054}
  [846] = {j1=-10.837, j2=61.047, j3=50.669, j4=-4.276, j5=74.455, j6=-11.635}
  [847] = {j1=-10.816, j2=61.558, j3=50.194, j4=-4.327, j5=74.827, j6=-11.207}
  [848] = {j1=-10.795, j2=62.071, j3=49.717, j4=-4.377, j5=75.209, j6=-10.774}
  [849] = {j1=-10.776, j2=62.585, j3=49.237, j4=-4.426, j5=75.600, j6=-10.335}
  [850] = {j1=-10.759, j2=63.101, j3=48.751, j4=-4.470, j5=76.002, j6=-9.893}
  [851] = {j1=-10.756, j2=63.192, j3=48.666, j4=-4.477, j5=76.074, j6=-9.815}
  [852] = {j1=-10.740, j2=63.700, j3=48.190, j4=-4.521, j5=76.469, j6=-9.378}
  [853] = {j1=-10.721, j2=64.262, j3=47.697, j4=-4.578, j5=76.853, j6=-8.908}
  [854] = {j1=-10.703, j2=64.748, j3=47.341, j4=-4.641, j5=77.063, j6=-8.538}
  [855] = {j1=-10.689, j2=65.070, j3=47.191, j4=-4.701, j5=77.054, j6=-8.337}
  [856] = {j1=-10.673, j2=65.326, j3=47.159, j4=-4.774, j5=76.890, j6=-8.222}
  [857] = {j1=-10.655, j2=65.527, j3=47.225, j4=-4.863, j5=76.593, j6=-8.179}
  [858] = {j1=-10.634, j2=65.682, j3=47.371, j4=-4.969, j5=76.186, j6=-8.195}
  [859] = {j1=-10.609, j2=65.800, j3=47.579, j4=-5.096, j5=75.690, j6=-8.257}
  [860] = {j1=-10.581, j2=65.889, j3=47.831, j4=-5.247, j5=75.126, j6=-8.350}
  [861] = {j1=-10.547, j2=65.957, j3=48.114, j4=-5.427, j5=74.513, j6=-8.460}
  [862] = {j1=-10.545, j2=65.984, j3=48.068, j4=-5.437, j5=74.606, j6=-8.388}
  [863] = {j1=-10.579, j2=65.916, j3=47.784, j4=-5.255, j5=75.219, j6=-8.279}
  [864] = {j1=-10.608, j2=65.828, j3=47.530, j4=-5.103, j5=75.784, j6=-8.186}
  [865] = {j1=-10.633, j2=65.711, j3=47.320, j4=-4.975, j5=76.281, j6=-8.125}
  [866] = {j1=-10.654, j2=65.557, j3=47.172, j4=-4.866, j5=76.690, j6=-8.110}
  [867] = {j1=-10.673, j2=65.357, j3=47.104, j4=-4.775, j5=76.988, j6=-8.154}
  [868] = {j1=-10.689, j2=65.102, j3=47.135, j4=-4.699, j5=77.153, j6=-8.271}
  [869] = {j1=-10.704, j2=64.782, j3=47.283, j4=-4.636, j5=77.163, j6=-8.473}
  [870] = {j1=-10.723, j2=64.296, j3=47.637, j4=-4.570, j5=76.954, j6=-8.846}
  [871] = {j1=-10.742, j2=63.735, j3=48.130, j4=-4.511, j5=76.570, j6=-9.317}
  [872] = {j1=-10.759, j2=63.227, j3=48.603, j4=-4.467, j5=76.177, j6=-9.753}
  [873] = {j1=-10.762, j2=63.138, j3=48.688, j4=-4.460, j5=76.107, j6=-9.830}
  [874] = {j1=-10.779, j2=62.623, j3=49.169, j4=-4.417, j5=75.709, j6=-10.270}
  [875] = {j1=-10.798, j2=62.112, j3=49.645, j4=-4.369, j5=75.323, j6=-10.706}
  [876] = {j1=-10.818, j2=61.602, j3=50.117, j4=-4.318, j5=74.947, j6=-11.137}
  [877] = {j1=-10.839, j2=61.092, j3=50.588, j4=-4.267, j5=74.579, j6=-11.562}
  [878] = {j1=-10.860, j2=60.583, j3=51.059, j4=-4.218, j5=74.218, j6=-11.980}
  [879] = {j1=-10.882, j2=60.071, j3=51.532, j4=-4.171, j5=73.862, j6=-12.392}
  [880] = {j1=-10.903, j2=59.557, j3=52.011, j4=-4.130, j5=73.509, j6=-12.796}
  [881] = {j1=-10.920, j2=59.106, j3=52.433, j4=-4.100, j5=73.203, j6=-13.141}
  [882] = {j1=-10.936, j2=58.657, j3=52.852, j4=-4.076, j5=72.908, j6=-13.474}
  [883] = {j1=-10.952, j2=58.215, j3=53.257, j4=-4.056, j5=72.634, j6=-13.790}
  [884] = {j1=-10.967, j2=57.786, j3=53.639, j4=-4.037, j5=72.391, j6=-14.087}
  [885] = {j1=-10.968, j2=57.770, j3=53.652, j4=-4.036, j5=72.383, j6=-14.097}
  [886] = {j1=-10.969, j2=57.788, j3=53.621, j4=-4.030, j5=72.436, j6=-14.066}
  [887] = {j1=-10.969, j2=57.803, j3=53.607, j4=-4.031, j5=72.444, j6=-14.056}
  [888] = {j1=-10.954, j2=58.235, j3=53.221, j4=-4.049, j5=72.693, j6=-13.756}
  [889] = {j1=-10.938, j2=58.681, j3=52.809, j4=-4.069, j5=72.975, j6=-13.435}
  [890] = {j1=-10.922, j2=59.133, j3=52.384, j4=-4.093, j5=73.278, j6=-13.097}
  [891] = {j1=-10.904, j2=59.588, j3=51.956, j4=-4.123, j5=73.591, j6=-12.748}
  [892] = {j1=-10.883, j2=60.104, j3=51.475, j4=-4.165, j5=73.949, j6=-12.341}
  [893] = {j1=-10.862, j2=60.615, j3=51.000, j4=-4.212, j5=74.306, j6=-11.928}
  [894] = {j1=-10.840, j2=61.125, j3=50.530, j4=-4.261, j5=74.666, j6=-11.510}
  [895] = {j1=-10.819, j2=61.633, j3=50.062, j4=-4.312, j5=75.031, j6=-11.086}
  [896] = {j1=-10.799, j2=62.141, j3=49.593, j4=-4.363, j5=75.404, j6=-10.658}
  [897] = {j1=-10.780, j2=62.651, j3=49.120, j4=-4.410, j5=75.787, j6=-10.224}
  [898] = {j1=-10.763, j2=63.164, j3=48.641, j4=-4.454, j5=76.182, j6=-9.786}
  [899] = {j1=-10.761, j2=63.253, j3=48.557, j4=-4.461, j5=76.252, j6=-9.709}
  [900] = {j1=-10.744, j2=63.760, j3=48.085, j4=-4.505, j5=76.644, j6=-9.273}
  [901] = {j1=-10.724, j2=64.321, j3=47.594, j4=-4.565, j5=77.027, j6=-8.802}
  [902] = {j1=-10.705, j2=64.806, j3=47.240, j4=-4.633, j5=77.236, j6=-8.428}
  [903] = {j1=-10.689, j2=65.126, j3=47.093, j4=-4.698, j5=77.225, j6=-8.224}
  [904] = {j1=-10.673, j2=65.381, j3=47.063, j4=-4.776, j5=77.059, j6=-8.106}
  [905] = {j1=-10.654, j2=65.580, j3=47.133, j4=-4.869, j5=76.761, j6=-8.062}
  [906] = {j1=-10.632, j2=65.733, j3=47.282, j4=-4.979, j5=76.352, j6=-8.076}
  [907] = {j1=-10.607, j2=65.849, j3=47.492, j4=-5.108, j5=75.854, j6=-8.137}
  [908] = {j1=-10.578, j2=65.937, j3=47.748, j4=-5.262, j5=75.289, j6=-8.229}
  [909] = {j1=-10.544, j2=66.004, j3=48.032, j4=-5.444, j5=74.676, j6=-8.337}
  [910] = {j1=-10.543, j2=66.023, j3=47.999, j4=-5.451, j5=74.742, j6=-8.286}
  [911] = {j1=-10.577, j2=65.957, j3=47.714, j4=-5.268, j5=75.355, j6=-8.178}
  [912] = {j1=-10.606, j2=65.869, j3=47.457, j4=-5.113, j5=75.921, j6=-8.087}
  [913] = {j1=-10.632, j2=65.754, j3=47.246, j4=-4.983, j5=76.419, j6=-8.027}
  [914] = {j1=-10.653, j2=65.601, j3=47.095, j4=-4.871, j5=76.829, j6=-8.013}
  [915] = {j1=-10.673, j2=65.403, j3=47.024, j4=-4.777, j5=77.128, j6=-8.059}
  [916] = {j1=-10.690, j2=65.149, j3=47.053, j4=-4.697, j5=77.295, j6=-8.177}
  [917] = {j1=-10.706, j2=64.830, j3=47.199, j4=-4.630, j5=77.306, j6=-8.382}
  [918] = {j1=-10.726, j2=64.345, j3=47.551, j4=-4.560, j5=77.098, j6=-8.757}
  [919] = {j1=-10.746, j2=63.785, j3=48.041, j4=-4.498, j5=76.716, j6=-9.229}
  [920] = {j1=-10.762, j2=63.279, j3=48.512, j4=-4.454, j5=76.326, j6=-9.665}
  [921] = {j1=-10.765, j2=63.190, j3=48.595, j4=-4.447, j5=76.257, j6=-9.741}
  [922] = {j1=-10.782, j2=62.678, j3=49.071, j4=-4.404, j5=75.865, j6=-10.178}
  [923] = {j1=-10.800, j2=62.170, j3=49.541, j4=-4.357, j5=75.486, j6=-10.609}
  [924] = {j1=-10.820, j2=61.664, j3=50.007, j4=-4.307, j5=75.117, j6=-11.036}
  [925] = {j1=-10.841, j2=61.157, j3=50.472, j4=-4.256, j5=74.754, j6=-11.458}
  [926] = {j1=-10.863, j2=60.649, j3=50.941, j4=-4.206, j5=74.396, j6=-11.876}
  [927] = {j1=-10.885, j2=60.137, j3=51.416, j4=-4.159, j5=74.037, j6=-12.290}
  [928] = {j1=-10.906, j2=59.619, j3=51.900, j4=-4.117, j5=73.676, j6=-12.700}
  [929] = {j1=-10.924, j2=59.162, j3=52.333, j4=-4.086, j5=73.357, j6=-13.053}
  [930] = {j1=-10.940, j2=58.706, j3=52.763, j4=-4.063, j5=73.046, j6=-13.396}
  [931] = {j1=-10.955, j2=58.258, j3=53.180, j4=-4.043, j5=72.757, j6=-13.721}
  [932] = {j1=-10.970, j2=57.824, j3=53.571, j4=-4.025, j5=72.503, j6=-14.024}
  [933] = {j1=-10.971, j2=57.808, j3=53.584, j4=-4.025, j5=72.495, j6=-14.034}
  [934] = {j1=-10.973, j2=57.828, j3=53.549, j4=-4.018, j5=72.552, j6=-14.001}
  [935] = {j1=-10.972, j2=57.844, j3=53.536, j4=-4.019, j5=72.560, j6=-13.990}
  [936] = {j1=-10.957, j2=58.280, j3=53.141, j4=-4.036, j5=72.819, j6=-13.685}
  [937] = {j1=-10.942, j2=58.731, j3=52.719, j4=-4.055, j5=73.115, j6=-13.356}
  [938] = {j1=-10.925, j2=59.190, j3=52.283, j4=-4.079, j5=73.433, j6=-13.009}
  [939] = {j1=-10.908, j2=59.650, j3=51.846, j4=-4.110, j5=73.758, j6=-12.652}
  [940] = {j1=-10.886, j2=60.169, j3=51.358, j4=-4.152, j5=74.123, j6=-12.239}
  [941] = {j1=-10.864, j2=60.681, j3=50.883, j4=-4.200, j5=74.483, j6=-11.824}
  [942] = {j1=-10.843, j2=61.189, j3=50.416, j4=-4.250, j5=74.841, j6=-11.407}
  [943] = {j1=-10.822, j2=61.695, j3=49.952, j4=-4.301, j5=75.201, j6=-10.986}
  [944] = {j1=-10.802, j2=62.200, j3=49.489, j4=-4.351, j5=75.567, j6=-10.560}
  [945] = {j1=-10.783, j2=62.706, j3=49.023, j4=-4.398, j5=75.943, j6=-10.131}
  [946] = {j1=-10.767, j2=63.216, j3=48.549, j4=-4.440, j5=76.332, j6=-9.696}
  [947] = {j1=-10.764, j2=63.305, j3=48.466, j4=-4.447, j5=76.402, j6=-9.620}
  [948] = {j1=-10.748, j2=63.810, j3=47.997, j4=-4.492, j5=76.790, j6=-9.185}
  [949] = {j1=-10.727, j2=64.369, j3=47.508, j4=-4.554, j5=77.171, j6=-8.713}
  [950] = {j1=-10.707, j2=64.854, j3=47.157, j4=-4.627, j5=77.378, j6=-8.336}
  [951] = {j1=-10.690, j2=65.172, j3=47.012, j4=-4.697, j5=77.366, j6=-8.131}
  [952] = {j1=-10.673, j2=65.426, j3=46.985, j4=-4.778, j5=77.199, j6=-8.011}
  [953] = {j1=-10.653, j2=65.624, j3=47.056, j4=-4.874, j5=76.899, j6=-7.965}
  [954] = {j1=-10.631, j2=65.776, j3=47.208, j4=-4.987, j5=76.489, j6=-7.978}
  [955] = {j1=-10.606, j2=65.891, j3=47.420, j4=-5.119, j5=75.991, j6=-8.037}
  [956] = {j1=-10.576, j2=65.978, j3=47.678, j4=-5.274, j5=75.425, j6=-8.128}
  [957] = {j1=-10.541, j2=66.044, j3=47.964, j4=-5.458, j5=74.812, j6=-8.235}
  [958] = {j1=-10.540, j2=66.063, j3=47.930, j4=-5.465, j5=74.879, j6=-8.183}
  [959] = {j1=-10.575, j2=65.997, j3=47.643, j4=-5.280, j5=75.492, j6=-8.077}
  [960] = {j1=-10.605, j2=65.911, j3=47.385, j4=-5.124, j5=76.058, j6=-7.987}
  [961] = {j1=-10.630, j2=65.796, j3=47.172, j4=-4.990, j5=76.556, j6=-7.929}
  [962] = {j1=-10.653, j2=65.645, j3=47.019, j4=-4.877, j5=76.967, j6=-7.916}
  [963] = {j1=-10.673, j2=65.448, j3=46.946, j4=-4.779, j5=77.267, j6=-7.964}
  [964] = {j1=-10.691, j2=65.195, j3=46.972, j4=-4.696, j5=77.435, j6=-8.084}
  [965] = {j1=-10.708, j2=64.877, j3=47.117, j4=-4.624, j5=77.448, j6=-8.291}
  [966] = {j1=-10.729, j2=64.393, j3=47.466, j4=-4.549, j5=77.242, j6=-8.668}
  [967] = {j1=-10.749, j2=63.835, j3=47.953, j4=-4.485, j5=76.863, j6=-9.141}
  [968] = {j1=-10.766, j2=63.331, j3=48.420, j4=-4.441, j5=76.476, j6=-9.575}
  [969] = {j1=-10.768, j2=63.242, j3=48.503, j4=-4.434, j5=76.408, j6=-9.651}
  [970] = {j1=-10.785, j2=62.734, j3=48.974, j4=-4.392, j5=76.021, j6=-10.084}
  [971] = {j1=-10.803, j2=62.229, j3=49.437, j4=-4.345, j5=75.649, j6=-10.512}
  [972] = {j1=-10.823, j2=61.726, j3=49.897, j4=-4.295, j5=75.285, j6=-10.935}
  [973] = {j1=-10.844, j2=61.221, j3=50.358, j4=-4.244, j5=74.928, j6=-11.355}
  [974] = {j1=-10.866, j2=60.714, j3=50.825, j4=-4.194, j5=74.571, j6=-11.772}
  [975] = {j1=-10.887, j2=60.201, j3=51.300, j4=-4.146, j5=74.210, j6=-12.188}
  [976] = {j1=-10.909, j2=59.681, j3=51.790, j4=-4.103, j5=73.841, j6=-12.604}
  [977] = {j1=-10.927, j2=59.219, j3=52.231, j4=-4.072, j5=73.511, j6=-12.964}
  [978] = {j1=-10.944, j2=58.757, j3=52.672, j4=-4.048, j5=73.187, j6=-13.315}
  [979] = {j1=-10.959, j2=58.303, j3=53.099, j4=-4.029, j5=72.885, j6=-13.648}
  [980] = {j1=-10.974, j2=57.865, j3=53.497, j4=-4.013, j5=72.622, j6=-13.955}
  [981] = {j1=-10.974, j2=57.850, j3=53.511, j4=-4.012, j5=72.613, j6=-13.966}
  [982] = {j1=-10.976, j2=57.871, j3=53.472, j4=-4.006, j5=72.675, j6=-13.930}
  [983] = {j1=-10.975, j2=57.887, j3=53.458, j4=-4.006, j5=72.683, j6=-13.919}
  [984] = {j1=-10.961, j2=58.327, j3=53.057, j4=-4.022, j5=72.951, j6=-13.610}
  [985] = {j1=-10.946, j2=58.783, j3=52.626, j4=-4.041, j5=73.258, j6=-13.274}
  [986] = {j1=-10.929, j2=59.247, j3=52.181, j4=-4.065, j5=73.588, j6=-12.920}
  [987] = {j1=-10.911, j2=59.711, j3=51.736, j4=-4.096, j5=73.923, j6=-12.556}
  [988] = {j1=-10.889, j2=60.233, j3=51.244, j4=-4.140, j5=74.295, j6=-12.138}
  [989] = {j1=-10.867, j2=60.746, j3=50.768, j4=-4.188, j5=74.657, j6=-11.721}
  [990] = {j1=-10.845, j2=61.253, j3=50.302, j4=-4.238, j5=75.013, j6=-11.303}
  [991] = {j1=-10.824, j2=61.756, j3=49.843, j4=-4.289, j5=75.369, j6=-10.884}
  [992] = {j1=-10.805, j2=62.258, j3=49.385, j4=-4.339, j5=75.730, j6=-10.462}
  [993] = {j1=-10.786, j2=62.762, j3=48.924, j4=-4.385, j5=76.099, j6=-10.036}
  [994] = {j1=-10.770, j2=63.269, j3=48.456, j4=-4.427, j5=76.483, j6=-9.605}
  [995] = {j1=-10.767, j2=63.357, j3=48.373, j4=-4.434, j5=76.552, j6=-9.529}
  [996] = {j1=-10.751, j2=63.860, j3=47.909, j4=-4.479, j5=76.936, j6=-9.096}
  [997] = {j1=-10.730, j2=64.418, j3=47.424, j4=-4.544, j5=77.313, j6=-8.624}
  [998] = {j1=-10.709, j2=64.900, j3=47.076, j4=-4.621, j5=77.518, j6=-8.245}
  [999] = {j1=-10.691, j2=65.218, j3=46.932, j4=-4.695, j5=77.505, j6=-8.038}
  [1000] = {j1=-10.673, j2=65.470, j3=46.907, j4=-4.780, j5=77.337, j6=-7.916}
  [1001] = {j1=-10.652, j2=65.667, j3=46.981, j4=-4.879, j5=77.036, j6=-7.868}
  [1002] = {j1=-10.630, j2=65.818, j3=47.134, j4=-4.994, j5=76.625, j6=-7.879}
  [1003] = {j1=-10.604, j2=65.932, j3=47.349, j4=-5.129, j5=76.127, j6=-7.937}
  [1004] = {j1=-10.574, j2=66.018, j3=47.607, j4=-5.286, j5=75.561, j6=-8.026}
  [1005] = {j1=-10.573, j2=66.038, j3=47.572, j4=-5.292, j5=75.629, j6=-7.974}
  [1006] = {j1=-10.603, j2=65.953, j3=47.313, j4=-5.134, j5=76.194, j6=-7.886}
  [1007] = {j1=-10.629, j2=65.839, j3=47.098, j4=-4.998, j5=76.693, j6=-7.830}
  [1008] = {j1=-10.652, j2=65.688, j3=46.944, j4=-4.881, j5=77.103, j6=-7.820}
  [1009] = {j1=-10.673, j2=65.492, j3=46.870, j4=-4.781, j5=77.404, j6=-7.869}
  [1010] = {j1=-10.692, j2=65.240, j3=46.893, j4=-4.694, j5=77.573, j6=-7.991}
  [1011] = {j1=-10.710, j2=64.923, j3=47.036, j4=-4.618, j5=77.588, j6=-8.200}
  [1012] = {j1=-10.732, j2=64.441, j3=47.382, j4=-4.538, j5=77.384, j6=-8.579}
  [1013] = {j1=-10.753, j2=63.885, j3=47.865, j4=-4.472, j5=77.009, j6=-9.051}
  [1014] = {j1=-10.769, j2=63.384, j3=48.327, j4=-4.427, j5=76.627, j6=-9.483}
  [1015] = {j1=-10.772, j2=63.295, j3=48.409, j4=-4.421, j5=76.559, j6=-9.559}
  [1016] = {j1=-10.788, j2=62.789, j3=48.875, j4=-4.379, j5=76.178, j6=-9.988}
  [1017] = {j1=-10.806, j2=62.288, j3=49.333, j4=-4.333, j5=75.811, j6=-10.413}
  [1018] = {j1=-10.826, j2=61.787, j3=49.789, j4=-4.283, j5=75.453, j6=-10.834}
  [1019] = {j1=-10.847, j2=61.284, j3=50.246, j4=-4.232, j5=75.099, j6=-11.252}
  [1020] = {j1=-10.868, j2=60.778, j3=50.710, j4=-4.182, j5=74.743, j6=-11.669}
  [1021] = {j1=-10.890, j2=60.265, j3=51.187, j4=-4.133, j5=74.381, j6=-12.087}
  [1022] = {j1=-10.912, j2=59.742, j3=51.681, j4=-4.089, j5=74.006, j6=-12.508}
  [1023] = {j1=-10.931, j2=59.276, j3=52.129, j4=-4.057, j5=73.666, j6=-12.875}
  [1024] = {j1=-10.947, j2=58.810, j3=52.579, j4=-4.033, j5=73.331, j6=-13.232}
  [1025] = {j1=-10.963, j2=58.351, j3=53.014, j4=-4.015, j5=73.019, j6=-13.571}
  [1026] = {j1=-10.977, j2=57.910, j3=53.417, j4=-4.000, j5=72.748, j6=-13.882}
  [1027] = {j1=-10.977, j2=57.895, j3=53.431, j4=-4.000, j5=72.739, j6=-13.893}
  [1028] = {j1=-10.979, j2=57.921, j3=53.383, j4=-3.992, j5=72.813, j6=-13.849}
  [1029] = {j1=-10.979, j2=57.937, j3=53.370, j4=-3.993, j5=72.822, j6=-13.839}
  [1030] = {j1=-10.965, j2=58.379, j3=52.963, j4=-4.007, j5=73.097, j6=-13.526}
  [1031] = {j1=-10.949, j2=58.840, j3=52.525, j4=-4.025, j5=73.414, j6=-13.184}
  [1032] = {j1=-10.933, j2=59.309, j3=52.071, j4=-4.049, j5=73.754, j6=-12.823}
  [1033] = {j1=-10.914, j2=59.776, j3=51.620, j4=-4.081, j5=74.098, j6=-12.453}
  [1034] = {j1=-10.892, j2=60.300, j3=51.124, j4=-4.126, j5=74.476, j6=-12.031}
  [1035] = {j1=-10.870, j2=60.814, j3=50.647, j4=-4.175, j5=74.840, j6=-11.611}
  [1036] = {j1=-10.848, j2=61.320, j3=50.183, j4=-4.226, j5=75.195, j6=-11.194}
  [1037] = {j1=-10.827, j2=61.821, j3=49.728, j4=-4.277, j5=75.547, j6=-10.776}
  [1038] = {j1=-10.808, j2=62.321, j3=49.275, j4=-4.326, j5=75.903, j6=-10.357}
  [1039] = {j1=-10.790, j2=62.821, j3=48.819, j4=-4.372, j5=76.267, j6=-9.934}
  [1040] = {j1=-10.774, j2=63.325, j3=48.356, j4=-4.413, j5=76.644, j6=-9.506}
  [1041] = {j1=-10.771, j2=63.413, j3=48.275, j4=-4.420, j5=76.712, j6=-9.431}
  [1042] = {j1=-10.755, j2=63.913, j3=47.815, j4=-4.465, j5=77.091, j6=-9.000}
  [1043] = {j1=-10.733, j2=64.468, j3=47.334, j4=-4.532, j5=77.464, j6=-8.529}
  [1044] = {j1=-10.711, j2=64.949, j3=46.990, j4=-4.614, j5=77.666, j6=-8.149}
  [1045] = {j1=-10.692, j2=65.265, j3=46.850, j4=-4.692, j5=77.650, j6=-7.939}
  [1046] = {j1=-10.673, j2=65.516, j3=46.827, j4=-4.782, j5=77.481, j6=-7.815}
  [1047] = {j1=-10.652, j2=65.712, j3=46.902, j4=-4.884, j5=77.180, j6=-7.765}
  [1048] = {j1=-10.628, j2=65.862, j3=47.057, j4=-5.002, j5=76.769, j6=-7.774}
  [1049] = {j1=-10.602, j2=65.976, j3=47.273, j4=-5.139, j5=76.271, j6=-7.829}
  [1050] = {j1=-10.572, j2=66.062, j3=47.532, j4=-5.299, j5=75.706, j6=-7.916}
  [1051] = {j1=-10.570, j2=66.085, j3=47.492, j4=-5.306, j5=75.784, j6=-7.857}
  [1052] = {j1=-10.601, j2=65.999, j3=47.232, j4=-5.145, j5=76.348, j6=-7.772}
  [1053] = {j1=-10.628, j2=65.886, j3=47.016, j4=-5.007, j5=76.845, j6=-7.718}
  [1054] = {j1=-10.651, j2=65.736, j3=46.861, j4=-4.887, j5=77.256, j6=-7.710}
  [1055] = {j1=-10.673, j2=65.541, j3=46.785, j4=-4.783, j5=77.557, j6=-7.762}
  [1056] = {j1=-10.693, j2=65.290, j3=46.806, j4=-4.691, j5=77.727, j6=-7.887}
  [1057] = {j1=-10.712, j2=64.975, j3=46.945, j4=-4.611, j5=77.743, j6=-8.097}
  [1058] = {j1=-10.735, j2=64.495, j3=47.287, j4=-4.526, j5=77.544, j6=-8.478}
  [1059] = {j1=-10.757, j2=63.942, j3=47.765, j4=-4.458, j5=77.174, j6=-8.949}
  [1060] = {j1=-10.773, j2=63.443, j3=48.222, j4=-4.412, j5=76.797, j6=-9.378}
  [1061] = {j1=-10.776, j2=63.355, j3=48.303, j4=-4.406, j5=76.730, j6=-9.453}
  [1062] = {j1=-10.791, j2=62.853, j3=48.763, j4=-4.365, j5=76.356, j6=-9.879}
  [1063] = {j1=-10.809, j2=62.354, j3=49.216, j4=-4.320, j5=75.994, j6=-10.300}
  [1064] = {j1=-10.829, j2=61.856, j3=49.667, j4=-4.270, j5=75.641, j6=-10.719}
  [1065] = {j1=-10.850, j2=61.355, j3=50.120, j4=-4.219, j5=75.290, j6=-11.136}
  [1066] = {j1=-10.871, j2=60.850, j3=50.583, j4=-4.168, j5=74.936, j6=-11.553}
  [1067] = {j1=-10.894, j2=60.336, j3=51.061, j4=-4.118, j5=74.571, j6=-11.974}
  [1068] = {j1=-10.916, j2=59.811, j3=51.559, j4=-4.073, j5=74.190, j6=-12.399}
  [1069] = {j1=-10.935, j2=59.341, j3=52.013, j4=-4.040, j5=73.843, j6=-12.772}
  [1070] = {j1=-10.952, j2=58.871, j3=52.470, j4=-4.016, j5=73.498, j6=-13.135}
  [1071] = {j1=-10.967, j2=58.408, j3=52.912, j4=-3.999, j5=73.176, j6=-13.479}
  [1072] = {j1=-10.981, j2=57.965, j3=53.320, j4=-3.985, j5=72.899, j6=-13.793}
  [1073] = {j1=-10.981, j2=57.949, j3=53.334, j4=-3.985, j5=72.890, j6=-13.804}
  [1074] = {j1=-10.983, j2=57.978, j3=53.282, j4=-3.978, j5=72.970, j6=-13.757}
  [1075] = {j1=-10.982, j2=57.994, j3=53.268, j4=-3.978, j5=72.979, j6=-13.747}
  [1076] = {j1=-10.969, j2=58.439, j3=52.858, j4=-3.990, j5=73.258, j6=-13.432}
  [1077] = {j1=-10.954, j2=58.902, j3=52.414, j4=-4.007, j5=73.583, j6=-13.086}
  [1078] = {j1=-10.937, j2=59.374, j3=51.954, j4=-4.031, j5=73.932, j6=-12.720}
  [1079] = {j1=-10.918, j2=59.845, j3=51.498, j4=-4.064, j5=74.283, j6=-12.344}
  [1080] = {j1=-10.895, j2=60.371, j3=50.998, j4=-4.111, j5=74.666, j6=-11.917}
  [1081] = {j1=-10.873, j2=60.885, j3=50.520, j4=-4.161, j5=75.031, j6=-11.495}
  [1082] = {j1=-10.851, j2=61.390, j3=50.058, j4=-4.212, j5=75.385, j6=-11.077}
  [1083] = {j1=-10.830, j2=61.890, j3=49.606, j4=-4.264, j5=75.735, j6=-10.661}
  [1084] = {j1=-10.811, j2=62.387, j3=49.157, j4=-4.313, j5=76.086, j6=-10.244}
  [1085] = {j1=-10.793, j2=62.884, j3=48.707, j4=-4.358, j5=76.445, j6=-9.824}
  [1086] = {j1=-10.777, j2=63.385, j3=48.250, j4=-4.398, j5=76.817, j6=-9.400}
  [1087] = {j1=-10.775, j2=63.473, j3=48.169, j4=-4.405, j5=76.883, j6=-9.325}
  [1088] = {j1=-10.758, j2=63.970, j3=47.715, j4=-4.450, j5=77.257, j6=-8.897}
  [1089] = {j1=-10.737, j2=64.522, j3=47.240, j4=-4.520, j5=77.623, j6=-8.427}
  [1090] = {j1=-10.713, j2=65.000, j3=46.901, j4=-4.607, j5=77.820, j6=-8.046}
  [1091] = {j1=-10.693, j2=65.315, j3=46.763, j4=-4.690, j5=77.802, j6=-7.834}
  [1092] = {j1=-10.673, j2=65.565, j3=46.743, j4=-4.783, j5=77.632, j6=-7.709}
  [1093] = {j1=-10.651, j2=65.760, j3=46.820, j4=-4.889, j5=77.331, j6=-7.655}
  [1094] = {j1=-10.627, j2=65.909, j3=46.976, j4=-5.011, j5=76.921, j6=-7.662}
  [1095] = {j1=-10.600, j2=66.023, j3=47.192, j4=-5.150, j5=76.424, j6=-7.714}
  [1096] = {j1=-10.569, j2=66.108, j3=47.452, j4=-5.312, j5=75.862, j6=-7.798}
  [1097] = {j1=-10.568, j2=66.132, j3=47.410, j4=-5.319, j5=75.940, j6=-7.738}
  [1098] = {j1=-10.599, j2=66.046, j3=47.151, j4=-5.156, j5=76.502, j6=-7.656}
  [1099] = {j1=-10.626, j2=65.933, j3=46.934, j4=-5.015, j5=76.998, j6=-7.606}
  [1100] = {j1=-10.650, j2=65.783, j3=46.779, j4=-4.892, j5=77.406, j6=-7.601}
  [1101] = {j1=-10.673, j2=65.589, j3=46.701, j4=-4.784, j5=77.707, j6=-7.655}
  [1102] = {j1=-10.694, j2=65.339, j3=46.721, j4=-4.689, j5=77.878, j6=-7.782}
  [1103] = {j1=-10.714, j2=65.025, j3=46.857, j4=-4.604, j5=77.897, j6=-7.995}
  [1104] = {j1=-10.738, j2=64.549, j3=47.193, j4=-4.514, j5=77.703, j6=-8.376}
  [1105] = {j1=-10.760, j2=63.999, j3=47.664, j4=-4.443, j5=77.340, j6=-8.845}
  [1106] = {j1=-10.777, j2=63.503, j3=48.116, j4=-4.398, j5=76.969, j6=-9.271}
  [1107] = {j1=-10.779, j2=63.416, j3=48.196, j4=-4.391, j5=76.903, j6=-9.346}
  [1108] = {j1=-10.795, j2=62.916, j3=48.651, j4=-4.352, j5=76.534, j6=-9.768}
  [1109] = {j1=-10.812, j2=62.420, j3=49.099, j4=-4.306, j5=76.178, j6=-10.187}
  [1110] = {j1=-10.832, j2=61.924, j3=49.545, j4=-4.257, j5=75.828, j6=-10.603}
  [1111] = {j1=-10.853, j2=61.425, j3=49.997, j4=-4.205, j5=75.480, j6=-11.019}
  [1112] = {j1=-10.874, j2=60.920, j3=50.458, j4=-4.154, j5=75.125, j6=-11.438}
  [1113] = {j1=-10.897, j2=60.406, j3=50.937, j4=-4.103, j5=74.759, j6=-11.861}
  [1114] = {j1=-10.920, j2=59.879, j3=51.438, j4=-4.056, j5=74.374, j6=-12.290}
  [1115] = {j1=-10.939, j2=59.407, j3=51.896, j4=-4.022, j5=74.020, j6=-12.667}
  [1116] = {j1=-10.956, j2=58.934, j3=52.358, j4=-3.999, j5=73.669, j6=-13.035}
  [1117] = {j1=-10.971, j2=58.469, j3=52.804, j4=-3.982, j5=73.341, j6=-13.383}
  [1118] = {j1=-10.984, j2=58.024, j3=53.215, j4=-3.970, j5=73.059, j6=-13.698}
  [1119] = {j1=-10.985, j2=58.008, j3=53.229, j4=-3.970, j5=73.050, j6=-13.709}
  [1120] = {j1=-10.986, j2=58.040, j3=53.172, j4=-3.963, j5=73.135, j6=-13.659}
  [1121] = {j1=-10.986, j2=58.055, j3=53.158, j4=-3.963, j5=73.145, j6=-13.648}
  [1122] = {j1=-10.973, j2=58.501, j3=52.747, j4=-3.974, j5=73.427, j6=-13.332}
  [1123] = {j1=-10.958, j2=58.966, j3=52.299, j4=-3.990, j5=73.757, j6=-12.984}
  [1124] = {j1=-10.941, j2=59.441, j3=51.836, j4=-4.014, j5=74.110, j6=-12.615}
  [1125] = {j1=-10.922, j2=59.913, j3=51.377, j4=-4.048, j5=74.466, j6=-12.235}
  [1126] = {j1=-10.899, j2=60.440, j3=50.875, j4=-4.095, j5=74.852, j6=-11.804}
  [1127] = {j1=-10.876, j2=60.955, j3=50.396, j4=-4.146, j5=75.220, j6=-11.380}
  [1128] = {j1=-10.854, j2=61.460, j3=49.935, j4=-4.199, j5=75.574, j6=-10.961}
  [1129] = {j1=-10.833, j2=61.958, j3=49.485, j4=-4.250, j5=75.922, j6=-10.545}
  [1130] = {j1=-10.814, j2=62.453, j3=49.040, j4=-4.300, j5=76.269, j6=-10.130}
  [1131] = {j1=-10.796, j2=62.948, j3=48.594, j4=-4.345, j5=76.623, j6=-9.712}
  [1132] = {j1=-10.781, j2=63.446, j3=48.142, j4=-4.384, j5=76.990, j6=-9.291}
  [1133] = {j1=-10.779, j2=63.533, j3=48.063, j4=-4.390, j5=77.055, j6=-9.217}
  [1134] = {j1=-10.762, j2=64.027, j3=47.614, j4=-4.436, j5=77.422, j6=-8.793}
  [1135] = {j1=-10.740, j2=64.575, j3=47.147, j4=-4.508, j5=77.781, j6=-8.325}
  [1136] = {j1=-10.715, j2=65.050, j3=46.814, j4=-4.600, j5=77.972, j6=-7.944}
  [1137] = {j1=-10.694, j2=65.363, j3=46.679, j4=-4.687, j5=77.952, j6=-7.731}
  [1138] = {j1=-10.673, j2=65.612, j3=46.661, j4=-4.785, j5=77.781, j6=-7.602}
  [1139] = {j1=-10.650, j2=65.807, j3=46.739, j4=-4.894, j5=77.480, j6=-7.546}
  [1140] = {j1=-10.626, j2=65.956, j3=46.895, j4=-5.019, j5=77.072, j6=-7.549}
  [1141] = {j1=-10.598, j2=66.069, j3=47.111, j4=-5.161, j5=76.578, j6=-7.598}
  [1142] = {j1=-10.567, j2=66.155, j3=47.371, j4=-5.325, j5=76.018, j6=-7.678}
  [1143] = {j1=-10.566, j2=66.179, j3=47.329, j4=-5.332, j5=76.097, j6=-7.618}
  [1144] = {j1=-10.597, j2=66.093, j3=47.069, j4=-5.167, j5=76.656, j6=-7.540}
  [1145] = {j1=-10.625, j2=65.980, j3=46.853, j4=-5.023, j5=77.149, j6=-7.493}
  [1146] = {j1=-10.650, j2=65.830, j3=46.698, j4=-4.897, j5=77.555, j6=-7.492}
  [1147] = {j1=-10.673, j2=65.636, j3=46.619, j4=-4.786, j5=77.855, j6=-7.549}
  [1148] = {j1=-10.695, j2=65.387, j3=46.637, j4=-4.686, j5=78.027, j6=-7.679}
  [1149] = {j1=-10.716, j2=65.075, j3=46.770, j4=-4.597, j5=78.048, j6=-7.893}
  [1150] = {j1=-10.741, j2=64.602, j3=47.100, j4=-4.502, j5=77.860, j6=-8.274}
  [1151] = {j1=-10.764, j2=64.056, j3=47.564, j4=-4.428, j5=77.505, j6=-8.740}
  [1152] = {j1=-10.780, j2=63.564, j3=48.009, j4=-4.383, j5=77.142, j6=-9.163}
  [1153] = {j1=-10.783, j2=63.477, j3=48.088, j4=-4.377, j5=77.077, j6=-9.237}
  [1154] = {j1=-10.798, j2=62.980, j3=48.538, j4=-4.338, j5=76.713, j6=-9.656}
  [1155] = {j1=-10.816, j2=62.486, j3=48.981, j4=-4.293, j5=76.361, j6=-10.072}
  [1156] = {j1=-10.835, j2=61.992, j3=49.425, j4=-4.244, j5=76.014, j6=-10.487}
  [1157] = {j1=-10.856, j2=61.494, j3=49.874, j4=-4.192, j5=75.667, j6=-10.904}
  [1158] = {j1=-10.878, j2=60.989, j3=50.335, j4=-4.139, j5=75.312, j6=-11.323}
  [1159] = {j1=-10.901, j2=60.474, j3=50.814, j4=-4.088, j5=74.944, j6=-11.748}
  [1160] = {j1=-10.924, j2=59.946, j3=51.317, j4=-4.039, j5=74.556, j6=-12.180}
  [1161] = {j1=-10.943, j2=59.473, j3=51.778, j4=-4.005, j5=74.199, j6=-12.561}
  [1162] = {j1=-10.960, j2=58.999, j3=52.242, j4=-3.981, j5=73.844, j6=-12.932}
  [1163] = {j1=-10.975, j2=58.533, j3=52.690, j4=-3.965, j5=73.513, j6=-13.281}
  [1164] = {j1=-10.988, j2=58.087, j3=53.102, j4=-3.955, j5=73.229, j6=-13.597}
  [1165] = {j1=-10.988, j2=58.071, j3=53.116, j4=-3.955, j5=73.220, j6=-13.607}
  [1166] = {j1=-10.990, j2=58.105, j3=53.055, j4=-3.948, j5=73.311, j6=-13.554}
  [1167] = {j1=-10.989, j2=58.121, j3=53.041, j4=-3.948, j5=73.320, j6=-13.543}
  [1168] = {j1=-10.977, j2=58.567, j3=52.629, j4=-3.957, j5=73.603, j6=-13.228}
  [1169] = {j1=-10.962, j2=59.032, j3=52.181, j4=-3.972, j5=73.934, j6=-12.879}
  [1170] = {j1=-10.945, j2=59.507, j3=51.717, j4=-3.996, j5=74.290, j6=-12.508}
  [1171] = {j1=-10.926, j2=59.981, j3=51.256, j4=-4.031, j5=74.648, j6=-12.126}
  [1172] = {j1=-10.902, j2=60.509, j3=50.753, j4=-4.080, j5=75.037, j6=-11.692}
  [1173] = {j1=-10.879, j2=61.024, j3=50.274, j4=-4.132, j5=75.405, j6=-11.266}
  [1174] = {j1=-10.857, j2=61.528, j3=49.813, j4=-4.185, j5=75.760, j6=-10.846}
  [1175] = {j1=-10.836, j2=62.026, j3=49.365, j4=-4.237, j5=76.107, j6=-10.429}
  [1176] = {j1=-10.817, j2=62.520, j3=48.922, j4=-4.286, j5=76.452, j6=-10.015}
  [1177] = {j1=-10.800, j2=63.013, j3=48.481, j4=-4.331, j5=76.803, j6=-9.599}
  [1178] = {j1=-10.785, j2=63.508, j3=48.034, j4=-4.369, j5=77.163, j6=-9.182}
  [1179] = {j1=-10.782, j2=63.594, j3=47.956, j4=-4.375, j5=77.228, j6=-9.108}
  [1180] = {j1=-10.766, j2=64.084, j3=47.514, j4=-4.421, j5=77.587, j6=-8.687}
  [1181] = {j1=-10.743, j2=64.628, j3=47.055, j4=-4.496, j5=77.938, j6=-8.222}
  [1182] = {j1=-10.717, j2=65.099, j3=46.728, j4=-4.593, j5=78.122, j6=-7.842}
  [1183] = {j1=-10.695, j2=65.410, j3=46.597, j4=-4.685, j5=78.099, j6=-7.627}
  [1184] = {j1=-10.673, j2=65.658, j3=46.580, j4=-4.786, j5=77.927, j6=-7.496}
  [1185] = {j1=-10.650, j2=65.853, j3=46.659, j4=-4.899, j5=77.628, j6=-7.437}
  [1186] = {j1=-10.624, j2=66.002, j3=46.814, j4=-5.027, j5=77.222, j6=-7.436}
  [1187] = {j1=-10.596, j2=66.116, j3=47.030, j4=-5.172, j5=76.731, j6=-7.481}
  [1188] = {j1=-10.564, j2=66.202, j3=47.289, j4=-5.338, j5=76.174, j6=-7.558}
  [1189] = {j1=-10.563, j2=66.227, j3=47.246, j4=-5.345, j5=76.255, j6=-7.497}
  [1190] = {j1=-10.595, j2=66.140, j3=46.988, j4=-5.177, j5=76.810, j6=-7.423}
  [1191] = {j1=-10.624, j2=66.026, j3=46.773, j4=-5.031, j5=77.299, j6=-7.380}
  [1192] = {j1=-10.649, j2=65.876, j3=46.618, j4=-4.902, j5=77.703, j6=-7.383}
  [1193] = {j1=-10.673, j2=65.682, j3=46.539, j4=-4.787, j5=78.001, j6=-7.444}
  [1194] = {j1=-10.696, j2=65.434, j3=46.555, j4=-4.684, j5=78.173, j6=-7.576}
  [1195] = {j1=-10.718, j2=65.124, j3=46.685, j4=-4.589, j5=78.197, j6=-7.791}
  [1196] = {j1=-10.745, j2=64.654, j3=47.008, j4=-4.490, j5=78.016, j6=-8.171}
  [1197] = {j1=-10.768, j2=64.113, j3=47.463, j4=-4.414, j5=77.671, j6=-8.634}
  [1198] = {j1=-10.784, j2=63.625, j3=47.902, j4=-4.368, j5=77.315, j6=-9.053}
  [1199] = {j1=-10.787, j2=63.538, j3=47.980, j4=-4.362, j5=77.251, j6=-9.126}
  [1200] = {j1=-10.801, j2=63.045, j3=48.424, j4=-4.324, j5=76.892, j6=-9.542}
  [1201] = {j1=-10.819, j2=62.553, j3=48.864, j4=-4.280, j5=76.544, j6=-9.957}
  [1202] = {j1=-10.838, j2=62.059, j3=49.306, j4=-4.230, j5=76.198, j6=-10.371}
  [1203] = {j1=-10.859, j2=61.562, j3=49.754, j4=-4.178, j5=75.851, j6=-10.788}
  [1204] = {j1=-10.881, j2=61.057, j3=50.215, j4=-4.125, j5=75.496, j6=-11.209}
  [1205] = {j1=-10.904, j2=60.542, j3=50.694, j4=-4.072, j5=75.126, j6=-11.636}
  [1206] = {j1=-10.928, j2=60.014, j3=51.197, j4=-4.022, j5=74.737, j6=-12.071}
  [1207] = {j1=-10.948, j2=59.540, j3=51.658, j4=-3.987, j5=74.379, j6=-12.454}
  [1208] = {j1=-10.964, j2=59.065, j3=52.123, j4=-3.963, j5=74.023, j6=-12.825}
  [1209] = {j1=-10.979, j2=58.600, j3=52.570, j4=-3.948, j5=73.691, j6=-13.174}
  [1210] = {j1=-10.991, j2=58.154, j3=52.981, j4=-3.940, j5=73.408, j6=-13.489}
  [1211] = {j1=-10.992, j2=58.139, j3=52.995, j4=-3.940, j5=73.399, j6=-13.499}
  [1212] = {j1=-10.993, j2=58.175, j3=52.930, j4=-3.932, j5=73.495, j6=-13.443}
  [1213] = {j1=-10.993, j2=58.191, j3=52.916, j4=-3.933, j5=73.504, j6=-13.432}
  [1214] = {j1=-10.981, j2=58.635, j3=52.506, j4=-3.939, j5=73.786, j6=-13.118}
  [1215] = {j1=-10.967, j2=59.100, j3=52.060, j4=-3.954, j5=74.116, j6=-12.770}
  [1216] = {j1=-10.950, j2=59.575, j3=51.597, j4=-3.978, j5=74.471, j6=-12.399}
  [1217] = {j1=-10.930, j2=60.048, j3=51.137, j4=-4.014, j5=74.828, j6=-12.016}
  [1218] = {j1=-10.906, j2=60.576, j3=50.634, j4=-4.065, j5=75.218, j6=-11.580}
  [1219] = {j1=-10.883, j2=61.091, j3=50.155, j4=-4.118, j5=75.588, j6=-11.152}
  [1220] = {j1=-10.860, j2=61.596, j3=49.694, j4=-4.172, j5=75.943, j6=-10.731}
  [1221] = {j1=-10.839, j2=62.093, j3=49.246, j4=-4.224, j5=76.290, j6=-10.313}
  [1222] = {j1=-10.820, j2=62.586, j3=48.805, j4=-4.273, j5=76.635, j6=-9.899}
  [1223] = {j1=-10.803, j2=63.077, j3=48.367, j4=-4.317, j5=76.982, j6=-9.485}
  [1224] = {j1=-10.788, j2=63.569, j3=47.926, j4=-4.355, j5=77.338, j6=-9.070}
  [1225] = {j1=-10.786, j2=63.655, j3=47.848, j4=-4.361, j5=77.401, j6=-8.998}
  [1226] = {j1=-10.770, j2=64.141, j3=47.414, j4=-4.407, j5=77.752, j6=-8.581}
  [1227] = {j1=-10.746, j2=64.680, j3=46.963, j4=-4.484, j5=78.093, j6=-8.120}
  [1228] = {j1=-10.719, j2=65.147, j3=46.644, j4=-4.586, j5=78.270, j6=-7.741}
  [1229] = {j1=-10.696, j2=65.457, j3=46.516, j4=-4.682, j5=78.243, j6=-7.524}
  [1230] = {j1=-10.673, j2=65.704, j3=46.501, j4=-4.787, j5=78.071, j6=-7.391}
  [1231] = {j1=-10.649, j2=65.898, j3=46.580, j4=-4.904, j5=77.774, j6=-7.328}
  [1232] = {j1=-10.623, j2=66.048, j3=46.735, j4=-5.034, j5=77.371, j6=-7.323}
  [1233] = {j1=-10.594, j2=66.163, j3=46.949, j4=-5.182, j5=76.884, j6=-7.364}
  [1234] = {j1=-10.562, j2=66.249, j3=47.207, j4=-5.351, j5=76.331, j6=-7.436}
  [1235] = {j1=-10.561, j2=66.274, j3=47.163, j4=-5.357, j5=76.413, j6=-7.374}
  [1236] = {j1=-10.593, j2=66.187, j3=46.906, j4=-5.187, j5=76.963, j6=-7.305}
  [1237] = {j1=-10.622, j2=66.072, j3=46.693, j4=-5.038, j5=77.448, j6=-7.267}
  [1238] = {j1=-10.649, j2=65.922, j3=46.539, j4=-4.906, j5=77.848, j6=-7.274}
  [1239] = {j1=-10.673, j2=65.727, j3=46.461, j4=-4.788, j5=78.144, j6=-7.338}
  [1240] = {j1=-10.697, j2=65.480, j3=46.476, j4=-4.681, j5=78.316, j6=-7.473}
  [1241] = {j1=-10.720, j2=65.171, j3=46.601, j4=-4.582, j5=78.344, j6=-7.690}
  [1242] = {j1=-10.748, j2=64.706, j3=46.917, j4=-4.478, j5=78.171, j6=-8.068}
  [1243] = {j1=-10.772, j2=64.170, j3=47.363, j4=-4.400, j5=77.836, j6=-8.527}
  [1244] = {j1=-10.788, j2=63.686, j3=47.794, j4=-4.354, j5=77.488, j6=-8.942}
  [1245] = {j1=-10.790, j2=63.600, j3=47.871, j4=-4.348, j5=77.425, j6=-9.014}
  [1246] = {j1=-10.805, j2=63.109, j3=48.310, j4=-4.310, j5=77.072, j6=-9.427}
  [1247] = {j1=-10.822, j2=62.619, j3=48.747, j4=-4.266, j5=76.725, j6=-9.841}
  [1248] = {j1=-10.841, j2=62.126, j3=49.188, j4=-4.217, j5=76.381, j6=-10.255}
  [1249] = {j1=-10.862, j2=61.629, j3=49.636, j4=-4.164, j5=76.033, j6=-10.673}
  [1250] = {j1=-10.884, j2=61.124, j3=50.097, j4=-4.110, j5=75.676, j6=-11.096}
  [1251] = {j1=-10.908, j2=60.609, j3=50.576, j4=-4.057, j5=75.306, j6=-11.525}
  [1252] = {j1=-10.932, j2=60.081, j3=51.079, j4=-4.005, j5=74.916, j6=-11.961}
  [1253] = {j1=-10.952, j2=59.608, j3=51.538, j4=-3.968, j5=74.559, j6=-12.344}
  [1254] = {j1=-10.969, j2=59.134, j3=52.000, j4=-3.944, j5=74.205, j6=-12.715}
  [1255] = {j1=-10.983, j2=58.670, j3=52.445, j4=-3.930, j5=73.877, j6=-13.062}
  [1256] = {j1=-10.994, j2=58.226, j3=52.853, j4=-3.925, j5=73.597, j6=-13.374}
  [1257] = {j1=-10.995, j2=58.210, j3=52.867, j4=-3.924, j5=73.588, j6=-13.384}
  [1258] = {j1=-10.997, j2=58.263, j3=52.774, j4=-3.915, j5=73.722, j6=-13.305}
  [1259] = {j1=-10.996, j2=58.278, j3=52.760, j4=-3.915, j5=73.731, j6=-13.295}
  [1260] = {j1=-10.985, j2=58.720, j3=52.355, j4=-3.920, j5=74.007, j6=-12.985}
  [1261] = {j1=-10.971, j2=59.182, j3=51.914, j4=-3.933, j5=74.332, j6=-12.640}
  [1262] = {j1=-10.954, j2=59.654, j3=51.455, j4=-3.957, j5=74.683, j6=-12.271}
  [1263] = {j1=-10.935, j2=60.126, j3=50.998, j4=-3.994, j5=75.037, j6=-11.888}
  [1264] = {j1=-10.910, j2=60.653, j3=50.497, j4=-4.046, j5=75.426, j6=-11.452}
  [1265] = {j1=-10.886, j2=61.168, j3=50.018, j4=-4.101, j5=75.796, j6=-11.022}
